DATA_BLOCK "Blok_Bledow"	// DB 119
VERSION : 0.1
  STRUCT
   Blad_Silnika_Adr_1 : BOOL ;	//Blad silnika o adresie 1 - rolki obrotnica bindownicy
   Blad_Silnika_Adr_2 : BOOL ;	//Blad silnika o adresie 2 - rolki wylot bindownicy
   Blad_Silnika_Adr_3 : BOOL ;	//Blad silnika o adresie 3 - rolki
   Blad_Silnika_Adr_4 : BOOL ;	//Blad silnika o adresie 4 - rolki
   Blad_Silnika_Adr_5 : BOOL ;	//Blad silnika o adresie 5 - rolki
   Blad_Silnika_Adr_6 : BOOL ;	//Blad silnika o adresie 6 - rolki
   Blad_Silnika_Adr_7 : BOOL ;	//Blad silnika o adresie 7 - rolki
   Blad_Silnika_Adr_8 : BOOL ;	//Blad silnika o adresie 8 - rolki
   Blad_Silnika_Adr_9 : BOOL ;	//Blad silnika o adresie 9 - rolki
   Blad_Silnika_Adr_10 : BOOL ;	//Blad silnika o adresie 10 - rolki
   Blad_Silnika_Adr_11 : BOOL ;	//Blad silnika o adresie 11 - rolki
   Blad_Silnika_Adr_12 : BOOL ;	//Blad silnika o adresie 12 - rolki
   Blad_Silnika_Adr_13 : BOOL ;	//Blad silnika o adresie 13 - rolki
   Blad_Silnika_Adr_14 : BOOL ;	//Blad silnika o adresie 14 - rolki
   Blad_Silnika_Adr_15 : BOOL ;	//Blad silnika o adresie 15 - silnik obrotnicy bindownicy
   Blad_Rygla_Adr_16 : BOOL ;	//Blad rygla drzwi o adresie 16
   Blad_Silnika_Adr_18 : BOOL ;	//Blad silnika o adresie 18 - silnik obrotnicy wyboru wlotu
   Blad_Silnika_Adr_20 : BOOL ;	//Blad silnika o adresie 20 - silnik obrotnicy etykietownicy
   Blad_Silnika_Adr_23 : BOOL ;	//Blad silnika o adresie 23 - rolki
   Blad_Silnika_Adr_24 : BOOL ;	//Blad silnika o adresie 24 - rolki
   Blad_Kurtyny_Adr_25 : BOOL ;	//Blad kurtyny wlotowej  adres 25
   Blad_Kurtyny_Adr_26 : BOOL ;	//Blad kurtyny wylotowej aders 26
   Blad_Not_Aus_27 : BOOL ;	//Blad Not Aus adres 27 - Not Aus szafa
   Blad_Not_Aus_28 : BOOL ;	//Blad Not Aus adres 28 - Not Aus poczatek lini
   Blad_Not_Aus_29 : BOOL ;	//Blad Not Aus adres 29 - Not Aus srodek lini
   Blad_Not_Aus_30 : BOOL ;	//Blad Not Aus adres 30 - Not Aus koniec lini
   Blad_Not_Aus_31 : BOOL ;	//Blad Not Aus adres 31 - Not Aus panel bindownicy
   Blad_Przek_Bezp_Bind : BOOL ;	//Strefa bezpieczenstwa rejonu bindownicy  niepotwierdzona(wejscie -I4.4)
   Ostrz_Bind_Blad : BOOL ;	//Blad ogolny bindownicy
   Ostrz_Bind_Nie_Cofnieta : BOOL ;	//Bindownica nie jest cofnieta
   Ostrz_Bind_Sygn_Bezp : BOOL ;	//Bindownica brak sygnalu bezpieczenstwa
   Ostrz_Bind_Nie_Jest_Auto : BOOL ;	//Bindownica nie jest w trybie automatycznym (wejscie -I2.4)
   Ostrz_Stol_Obr_Foto : BOOL ;	//Blad fotokomorek stolu obrotowego
   Ostrz_Obr_Stol_Obr_Pozyc : BOOL ;	//Stol obrotowy nie jest w pozycji 0
   Ostrz_Pokr_Foto_Tas_1 : BOOL ;	//Niewlasciwe Pokrycie fotkomorek na tasmie 1 (Przejedz do przodu w recznym )
   Ostrz_Pokr_Foto_Tas_2 : BOOL ;	//Niewlasciwe Pokrycie fotkomorek na tasmie 2 (Przejedz do przodu w recznym )
   Ostrz_Pokr_Foto_Obr : BOOL ;	//Niewlasciwe Pokrycie fotkomorek na obrotnicy (Przejedz do przodu w recznym )
   Ostrz_Pokr_Foto_Tas_4 : BOOL ;	//Niewlasciwe Pokrycie fotkomorek na tasmie 4 (Przejedz do przodu w recznym )
   Blad_Krok_1 : BOOL ;	//Blad kroku nr 1 (Przekrokczony czas jazdy  na zadana pozycje)
   Blad_Krok_2 : BOOL ;	//Blad kroku nr 2 (Przekrokczony czas szukania srodka palety)
   Blad_Krok_3 : BOOL ;	//Blad kroku nr 3 (Przekrokczony czas pozycjonowania palety lewo/prawo)
   Blad_Krok_4 : BOOL ;	//Blad kroku nr 4 (Przekrokczony czas strzalu bindownicy)
   Blad_Krok_5 : BOOL ;	//Blad kroku nr 5 (Przekrokczony czas czasu postoju)
   Blad_Krok_6 : BOOL ;	//Blad kroku nr 6 (Przekrokczony czas powrotu lewo/prawo)
   Alarm_Obr_Stol_Obr_Pozyc : BOOL ;	//Stol obrotowy nie jest w pozycji 0
   Alarm_Bind_Nie_Cofinieta : BOOL ;	//Bindownica nie cofnieta lub brak zezwolenia  (cofnij ramie do tylu)
   Alarm_Bind_Sygn_Bezp : BOOL ;	//Bindownica brak sygnalu bezpieczenstwa
   rez3 : BOOL ;	//rez 3
   rez_6_0 : BOOL ;	//rez_6_0
   Alarm_Pokr_Foto_Tas_1 : BOOL ;	//Niewlasciwe Pokrycie fotkomorek na tasmie 1 (Przejedz do przodu w recznym )
   Alarm_Pokr_Foto_Tas_2 : BOOL ;	//Niewlasciwe Pokrycie fotkomorek na tasmie 2 (Przejedz do przodu w recznym )
   Alarm_Pokr_Foto_Tas_4 : BOOL ;	//Niewlasciwe Pokrycie fotkomorek na tasmie 4 (Przejedz do przodu w recznym )
   Alarm_Pokr_Foto_Obr : BOOL ;	//Niewlasciwe Pokrycie fotkomorek na obrotnicy przy braku cyklu
   Alarm_Bind_Nie_Jest_Auto : BOOL ;	//Bindownica nie jest w trybie automatycznym (wejscie -I2.4)
   Alarm_Bind_Blad : BOOL ;	//Blad ogolny bindownicy
   rez_6_7 : BOOL ;	//rez_6_7
   Ostrz_Prasa_Nie_W_Gorze : BOOL ;	//Zlamywak dekli nie jest u gory I2.6
   rez_7_1 : BOOL ;	//rez_7_1
   rez_7_2 : BOOL ;	//rez_7_2
   rez_7_3 : BOOL ;	//rez_7_3
   rez_7_4 : BOOL ;	//rez_7_4
   rez_7_5 : BOOL ;	//rez_7_5
   Ostrz_Wozek_Przy_Przen : BOOL ;	//Wozek widlowy przy przenosniku (i2.7)
   Ostrz_C_Bind_Foto_Pokr : BOOL ;	//Pokrycie fotokomorek podczas cyklu bindowania
   Ostrz_C_Bind_Poz_Bindow : BOOL ;	//Pozycja bindownicy podczas bindowania
   rez_8_1 : BOOL ;	//rez_8_1
   rez_8_2 : BOOL ;	//rez_8_2
   rez_8_3 : BOOL ;	//rez_8_3
   rez_8_4 : BOOL ;	//rez_8_4
   rez_8_5 : BOOL ;	//rez_8_5
   rez_8_6 : BOOL ;	//rez_8_6
   rez_8_7 : BOOL ;	//rez_8_7
   rez_9_0 : BOOL ;	//rez_9_0
   rez_9_1 : BOOL ;	//rez_9_1
   rez_9_2 : BOOL ;	//rez_9_2
   rez_9_3 : BOOL ;	//rez_9_3
   rez_9_4 : BOOL ;	//rez_9_4
   rez_9_5 : BOOL ;	//rez_9_5
   rez_9_6 : BOOL ;	//rez_9_6
   rez_9_7 : BOOL ;	//rez_9_7
   rez_int_bl : INT ;
   rez_int_bl_2 : INT ;
  END_STRUCT ;	
BEGIN
END_DATA_BLOCK

DATA_BLOCK "DB_HMI"	// DB 120
VERSION : 0.1
  STRUCT
   HMI_IN : STRUCT 	//Zmienne wchodzace do HMI nie nadpisywane W HMI (100 bajtow)
    Tryb_Reczny : BOOL ;	//Tryb Reczny
    Tryb_Auto : BOOL ;	//Tryb Auto
    Pozycja_0_st : BOOL ;	//Obrotnica Pozycja 0 st
    Pozycja_90_st : BOOL ;	//Obrotnica Pozycja 90 st
    Pozycja_180_st : BOOL ;	//Obrotnica Pozycja 180 st
    Pozycja_270_st : BOOL ;	//Obrotnica Pozycja 270 st
    Foto_Tasma_1_Tyl : BOOL ;	//foto tylne na bandzie wlotowej
    Foto_Tasma_1_Przod : BOOL ;	//foto przednie bandzie wlotowej
    Foto_Tasma_2_Tyl : BOOL ;	//foto tylne na bandzie wlotowej 2
    Foto_Tasma_2_Przod : BOOL ;	//foto przednie na bandzie wlotowej 2
    Foto_Obrotnica_3_Tyl : BOOL ;	//foto tylne na obrotnicy 3
    Foto_Obrotnica_3_Przod : BOOL ;	//foto przednie na obrotnicy 3
    Foto_Tasma_4_Tyl : BOOL ;	//foto tylne na bandzie wylotowej 4
    Foto_Tasma_4_Przod : BOOL ;	//foto przednie na bandzie wlotowej 4
    Motor_Tasma_1_Tyl : BOOL ;	//motor tasma 1 tyl
    Motor_Tasma_1_Przod : BOOL ;	//motor tasma 1 przod
    Motor_Tasma_2_Tyl : BOOL ;	//motor tasma 2 tyl
    Motor_Tasma_2_Przod : BOOL ;	//motor tasma 2 przod
    Motor_Tasma_3_Tyl : BOOL ;	//motor tasma obrotnica 3 tyl
    Motor_Tasma_3_Przod : BOOL ;	//motor tasma obrotnica 3 przod
    Motor_Obrotnica_3_CW : BOOL ;	//motor obrotnica 3 clock wise
    Motor_Obrotnica_3_CCW : BOOL ;	//motor obrotnica 3 counter clock wise
    Motor_Tasma_4_Przod : BOOL ;	//motor tasma obrotnica 4 tyl
    Motor_Tasma_4_Tyl : BOOL ;	//motor tasma obrotnica 4 przod
    Kurtyna_Wlot_Ok : BOOL ;	//kurtyna na wlocie ok
    Kurtyna_Wylot_Ok : BOOL ;	//kurtyna na wylocie ok
    Wybrano_TP_Przelot : BOOL ;	//wybrano tryb pracy przelot
    Wybrano_TP_Wiazanie_Wzdl : BOOL ;	//wybrano tryb pracy wiazanie wzdluzne
    Wybrano_TP_Wiazanie_Pop : BOOL ;	//wybrano tryb pracy wiazanie poprzeczne
    Wybrano_TP_Wiazanie_Krzy : BOOL ;	//wybrano tryb pracy wiazanie krzyzowe
    Czujnik_Ham_0_St : BOOL ;	//fotokomorka hamowania obrotnicy do kata 0st
    Czujnik_0_St : BOOL ;	//fotokomorka zatrzymania obrotnicy przy kacie 0st
    Czujnik_Ham_90_St : BOOL ;	//fotokomorka hamowania obrotnicy do kata 90st
    Czujnik_90_St : BOOL ;	//fotokomorka zatrzymania obrotnicy przy kacie 90st
    Czujnik_Ham_180_St : BOOL ;	//fotokomorka hamowania obrotnicy do kata 180st
    Czujnik_180_St : BOOL ;	//fotokomorka zatrzymania obrotnicy przy kacie 180st
    Czujnik_Ham_270_St : BOOL ;	//fotokomorka hamowania obrotnicy do kata 270st
    Czujnik_270_St : BOOL ;	//fotokomorka zatrzymania obrotnicy przy kacie 270st
    Interfefs_B_do_TP_B1 : BOOL ;	//obwod bezpieczenstwa bindownicy
    Interfefs_B_do_TP_B2 : BOOL ;	//polozenie podstawowe bindownicy
    Interfefs_B_do_TP_B3 : BOOL ;	//start/zakonczenie wiazania
    Interfefs_B_do_TP_B5 : BOOL ;	//blad bindownicy
    Interfefs_TP_do_B_TP1 : BOOL ;	//obwod bezpieczenstwa tasmociagow
    Interfefs_TP_do_B_TP2 : BOOL ;	//zezwolenie na prace bindownicy
    Interfefs_TP_do_B_TP3 : BOOL ;	//start wiazania
    PB_Strefa_bezpieczenstwa : BOOL ;	//przycisk zalaczenie Strefy bezpieczenstwa
    PB_Reczny : BOOL ;	//przycisk trybu reczny
    PB_Auto : BOOL ;	//przycisk auto
    PB_Reset : BOOL ;	//przycisk reset
    PB_Stop : BOOL ;	//przycisk stop
    PB_Cykl_Start : BOOL ;	//przycisk start cyklu
    PB_Tasma1_Tyl : BOOL ;	//przycisk tasma 1 do tylu
    PB_Tasma1_Przod : BOOL ;	//przycisk tasma 1 do przodu
    PB_Tasma2_Tyl : BOOL ;	//przycisk tasma 2 do tylu
    PB_Tasma2_Przod : BOOL ;	//przycisk tasma 2 do przodu
    PB_Tasma3_Tyl : BOOL ;	//przycisk tasma 3 do tylu
    PB_Tasma3_Przod : BOOL ;	//przycisk tasma 3 do przodu
    PB_Tasma4_Tyl : BOOL ;	//przycisk tasma 4 do tylu
    PB_Tasma4_Przod : BOOL ;	//przycisk tasma 4 do przodu
    PB_Tasma3_Obr_CW : BOOL ;	//przycisk obrotnica w prawo
    PB_Tasma3_Obr_CCW : BOOL ;	//przycisk obrotnica w lewo
    Lampka_Blad_Bind : BOOL ;	//lamka bledu bindownicy
    Lampka_Strzal_Tasmy : BOOL ;	//lampka wystrzalu tasmy
    Lampka_Strefa_Bezp : BOOL ;	//lampka przycisku strefy bezpieczenstwa
    Lampka_PB_Reczny : BOOL ;	//lampka przycisku trybu recznego
    Lampka_PB_Auto : BOOL ;	//lampka przycisku trybu auto
    Lampka_PB_Reset : BOOL ;	//lampka przycisku reset
    Lampka_PB_Stop : BOOL ;	//lampka przycisku stop
    Lampka_PB_Cykl_Start : BOOL ;	//lampka przycisku start
    Paleta_na_Tasmie_1 : BOOL ;	//znacznik palety na tasmie 1
    Paleta_na_Tasmie_2 : BOOL ;	//znacznik palety na tasmie 2
    Paleta_na_Tasmie_3_0_180 : BOOL ;	//znacznik palety na tasmie 3 przy kacie 0 lub 180st
    Paleta_na_Tasmie_3_90_27 : BOOL ;	//znacznik palety na tasmie 3 przy kacie 90 lub 270st
    Paleta_na_Tasmie_4 : BOOL ;	//znacznik palety na tasmie 4
    Paleta_na_Tasmie_1_T : BOOL ;	//znacznik palety na tasmie 1 wjazd
    Paleta_na_Tasmie_1_P : BOOL ;	//znacznik palety na tasmie 1 wyjazd
    Paleta_na_Tasmie_2_T : BOOL ;	//znacznik palety na tasmie 2 wjazd
    Paleta_na_Tasmie_2_P : BOOL ;	//znacznik palety na tasmie 2 wyjazd
    Paleta_na_Tasmie_3_T : BOOL ;	//znacznik palety na tasmie 3 wjazd
    Paleta_na_Tasmie_3_P : BOOL ;	//znacznik palety na tasmie 3 wyjazd
    Paleta_na_Tasmie_4_T : BOOL ;	//znacznik palety na tasmie 4 wjazd
    Paleta_na_Tasmie_4_P : BOOL ;	//znacznik palety na tasmie 4 wyjazd
    Rygiel : BOOL ;	//znacznik rygla drzwi
    Blad : BOOL ;	//Znacznik bledu
    Linia_transportowa_praca : BOOL ;	//Znacznik pracy calej linii transportowej
    Interfefs_B_do_TP_B4 : BOOL ;	//tryb pracy bindownicy: Auto(1) Reczny(0)
    Krok_1 : BOOL ;	//krok 1 trybu pracy
    Krok_2 : BOOL ;	//krok 2 trybu pracy
    Krok_3 : BOOL ;	//krok 3 trybu pracy
    Krok_4 : BOOL ;	//krok 4 trybu pracy
    Krok_5 : BOOL ;	//krok 5 trybu pracy
    Krok_6 : BOOL ;	//krok 6 trybu pracy
    Znacznik_Migania_Bledu : BOOL ;	//znacznik migania bledu
    Czujnik_Prasa : BOOL ;	//czujnik prasy s 22
    Stan_Zaworu : BOOL ;
    Gender_Jest_Online : BOOL ;	//Zalacz Gender do lini Gender Feeder
    Gender_Jest_OFFline : BOOL ;	//Odlacz Gender do lini Gender Feeder
    Obr_Gender_Wzdluz : BOOL ;
    Obr_za_Genderem_wzdluz : BOOL ;
    Obr_za_Foliarka_wzdluz : BOOL ;
    Obr_Gender_ukryj : BYTE ;
    Obr_za_Genderem_ukryj : BYTE ;
    Obr_za_Foliarka_ukryj : BYTE ;
    Tablica_IN_bool : ARRAY  [1 .. 10 ] OF BOOL  := FALSE;
    Tablica_IN_Byte : ARRAY  [1 .. 2 ] OF BYTE  := B#16#0;
    input_0 : BYTE ;
    input_1 : BYTE ;
    input_2 : BYTE ;
    input_3 : BYTE ;
    output_0 : BYTE ;
    output_1 : BYTE ;
    output_2 : BYTE ;
    output_3 : BYTE ;
    input_8 : BYTE ;
    input_9 : BYTE ;
    input_10 : BYTE ;
    input_11 : BYTE ;
    Tablica_IN_DWORD : ARRAY  [1 .. 4 ] OF DWORD ;
    NR_Kroku : DINT ;	//Numer kroku
    Aktualna_Data : DATE_AND_TIME ;
    Tablica_IN_INT : ARRAY  [1 .. 18 ] OF INT ;
    tryb_wiaz : INT ;	//znacznik wyboru trybu wiazania
    INT_Liczba_Akt_Kroku : INT ;	//znacznik wyboru aktualnie wykonywanego kroku
   END_STRUCT ;
   HMI_OUT : STRUCT 	//Zmienne wychodzace z HMI Nie nadpisywane w sterowniku od 100 bajta
    Wybor_2_Lap : BOOL ;	//Wybranie 2 lap
    Wybor_4_Lap : BOOL ;	//Wybranie 4 lap
    Start_Lini_z_OP : BOOL ;	//start calej lini z HMI
    Stop_Lini_z_OP : BOOL ;	//stop calej lini z HMI
    Wyzwolenie_Wyjazdu : BOOL ;	//wyzwolenie wyjazdu palety na stanowisku bindujacym (tylko w auto)
    Przycisk_Test_Lampek : BOOL ;	//przycisk test lampek
    Przycisk_Reset_Bledow : BOOL ;	//Przycisk resetowania bledow na panelu HMI
    Przycisk_Pozycjonowanie : BOOL ;	//Przycisk HMI do pozycjonowania palety
    H_Zalacz_Zawor_Prasa : BOOL ;	//Zalacz zawor prasa
    H_Zezwl_Ekran_Prasa : BOOL ;	//Zezwolenie na prase reczny
    PB_Gender_ONline : BOOL ;	//Przycisk Gender jest online z linia transportowa
    PB_Gender_OFFline : BOOL ;	//Przycisk Gender jest offline z linia transportowa
    Tablica_OUT_Bool : ARRAY  [1 .. 144 ] OF BOOL ;
    Tablina_OUT_INT : ARRAY  [1 .. 40 ] OF INT ;
   END_STRUCT ;
   HMI_IN_OUT : STRUCT 	//Zmienne nadpisywane w sterowniku i w HMI od 200 bajta
    Rezerwa_IN_Out_1 : BOOL ;
    Tp_Przelot : BOOL ;	//Tryb Pracy Przelot
    Tp_Wiazanie_Poprzeczne : BOOL ;	//Tryb Pracy Wiazanie poprzeczne
    Tp_Wiazanie_Wzdluzne : BOOL ;	//Tryb Pracy Wiazanie wzduzne
    Tp_Wiazanie_Pop_Wzdl : BOOL ;	//Tryb Pracy Wiaznie Poprzeczne i wzdluzne
    Tp_Pozycjonowanie : BOOL ;	//Tryb Pracy Pozycjonowanie Palety zalaczone
    Test_Lampek : BOOL ;	//Test Lampek
    Reset_bledow : BOOL ;	//Reset Bledow
    Zlamywak_Dekl : BOOL ;	//lamanie dekli
    Tablica_IN_OUT_Bool : ARRAY  [1 .. 144 ] OF BOOL ;
    Tablica_IN_OUT_INT : ARRAY  [1 .. 40 ] OF INT ;
    Wybor_trybu_pracy : BYTE ;
   END_STRUCT ;
  END_STRUCT ;	
BEGIN
   HMI_IN.Foto_Obrotnica_3_Przod := TRUE;
   HMI_IN.Czujnik_0_St := TRUE;
END_DATA_BLOCK

DATA_BLOCK "Kom_Shuttle"	// DB 205
VERSION : 0.1
  STRUCT
   OUT : STRUCT 	//Temporary placeholder variable
    Bit_Com_Odbieranie : BOOL ;
    Auto_Reczny_Gender : BOOL ;	//1-auto , 0- reczny
    Marka_Bezp_Gender : BOOL ;
    Linia_Gender_Online : BOOL ;	//Linia Gender odbiera palety z shuttle
    Blad_Lini_Gender : BOOL ;	//Linia Gender jest w bledzie
    Res_0_5 : BOOL ;
    PB_Auto : BOOL ;
    PB_Reczny : BOOL ;
    PB_Banda_Wozek_Przod : BOOL ;
    PB_Banda_Wozek_Tyl : BOOL ;
    Banda_1_Gen_Zez_Do_Pop : BOOL ;	//banda gender zezwolenie do porzedniej
    Banda_1_Gen_Pal_Dost : BOOL ;	//Paleta dostarczona
    Banda_1_Gen_Zez_R_Do_Pop : BOOL ;	//zezwolenie reczny do poprzedniej
    Res_1_5 : BOOL ;
    Res_1_6 : BOOL ;
    Res_1_7 : BOOL ;
    Bindownica_Agregat_Auto : BOOL ;	//Agregat bindownicy jest w auto
    Res_2_1 : BOOL ;
    Res_2_2 : BOOL ;
    Res_2_3 : BOOL ;
    Res_2_4 : BOOL ;
    Res_2_5 : BOOL ;
    Res_2_6 : BOOL ;
    Res_2_7 : BOOL ;
    Res_3_0 : BOOL ;
    Res_3_1 : BOOL ;
    Res_3_2 : BOOL ;
    Res_3_3 : BOOL ;
    Res_3_4 : BOOL ;
    Res_3_5 : BOOL ;
    Res_3_6 : BOOL ;
    Res_3_7 : BOOL ;
    Zmienna_DINT : DINT ;
   END_STRUCT ;
   IN : STRUCT 	//Temporary placeholder variable
    Bit_Com_Odbieranie : BOOL ;
    Auto_Reczny_Shuttle : BOOL ;	//1-auto , 0- reczny
    Marka_Bezp_Shuttle : BOOL ;
    Wymuszenie_Online : BOOL ;	//Wymuszenie Lini gender online
    Wymuszenie_Offline : BOOL ;	//Wymuszenie Lini gender offline (wykorzystanie wozka widlowego)
    Wozek_Na_Pozycji_Gender : BOOL ;	//Wozek znajduje sie na pozycji
    Wozek_Zasprzeglony : BOOL ;
    Res_0_7 : BOOL ;	//Przycisk reczny
    Wozek_Zab_do_Nast : BOOL ;	//Wozek zabierz do nastepnej
    Wozek_Zez_R_do_Nast : BOOL ;	//Wozek zezwolenie reczny do nastepnej
    Foto_Wozek_Przod : BOOL ;	//Foto Wozek Przod
    Foto_Wozek_Tyl : BOOL ;	//Foto Wozek Tyl
    Motor_Wozek_Tyl : BOOL ;	//Motor wozek tyl
    Motor_Wozek_Przod : BOOL ;	//Motor wozek przod
    Res_1_6 : BOOL ;
    Res_1_7 : BOOL ;
    Res_2_0 : BOOL ;
    Res_2_1 : BOOL ;
    Res_2_2 : BOOL ;
    Res_2_3 : BOOL ;
    Res_2_4 : BOOL ;
    Res_2_5 : BOOL ;
    Res_2_6 : BOOL ;
    Res_2_7 : BOOL ;
    Res_3_0 : BOOL ;
    Res_3_1 : BOOL ;
    Res_3_2 : BOOL ;
    Res_3_3 : BOOL ;
    Res_3_4 : BOOL ;
    Res_3_5 : BOOL ;
    Res_3_6 : BOOL ;
    Res_3_7 : BOOL ;
    Zmienna_DINT : DINT ;
   END_STRUCT ;
  END_STRUCT ;	
BEGIN
END_DATA_BLOCK

DATA_BLOCK "Rejestr Band"	// DB 310
VERSION : 0.1
  STRUCT
   Tasma_Wozek_0 : DINT ;	//Wartosc tasmy wozek
   Tasma_Gender_1 : DINT ;	//Wartosc tasmy gender
   Tasma_Gender_2 : DINT ;	//Wartosc tasmy gender
   Tasma_Gender_Obr_3 : DINT ;	//Wartosc tasmy gender obrot
   Tasma_Gender_4 : DINT ;	//Wartosc tasmy gender wylot
   Tasma_Transp_Obr_4 : DINT ;	//Wartosc tasmy obrotnicy 1 transportera
   Tasma_Transp_3 : DINT ;	//Tasma transportowa wlot 2
   Tasma_Transp_5 : DINT ;	//Tasma transportowa 5
   Tasma_Transp_6 : DINT ;	//Tasma transportowa 6
   Tasma_Transp_7 : DINT ;	//Tasma transportowa 7
   Tasma_Transp_8 : DINT ;	//Tasma transportowa 8
   Tasma_Transp_9 : DINT ;	//Tasma transportowa 9
   Tasma_Transp_10_Fol : DINT ;	//Tasma transportowa 10 wspolnsna z foliarka
   Tasma_Transp_4_Fol : DINT ;	//Tasma transportowa virtual 4
   Tasma_Transp_Obr_Fol : DINT ;	//Tasma transportowa obrotnica virtual 5
   Tasma_Transp_6_Fol : DINT ;	//Tasma za obrotnica virtulal 6
   Tasma_Transp_11_Fol : DINT ;	//Tasma transportowa 11 wspolna z foliarka
   Tasma_Transp_12 : DINT ;	//Tasma transportowa wlot 12
   Tasma_Transp_Obr_13 : DINT ;	//Tasma transportowa 13 obrotnica
   Tasma_Wysjsciowa_14 : DINT ;	//Tasma transportowa 14 wylot
  END_STRUCT ;	
BEGIN
END_DATA_BLOCK

DATA_BLOCK "Rejestr_Band_HMI"	// DB 311
VERSION : 0.1
  STRUCT
   Tasma_Wozek_0_HMI : DINT ;	//Wartosc tasmy wozek
   Tasma_Gender_1_HMI : DINT ;	//Wartosc tasmy gender
   Tasma_Gender_2_HMI : DINT ;	//Wartosc tasmy gender
   Tasma_Gender_Obr_3_HMI : DINT ;	//Wartosc tasmy gender obrot
   Tasma_Gender_4_HMI : DINT ;	//Wartosc tasmy gender wylot
   Tasma_Transp_Obr_4_HMI : DINT ;	//Wartosc tasmy obrotnicy 1 transportera
   Tasma_Transp_3_HMI : DINT ;	//Tasma transportowa wlot 2
   Tasma_Transp_5_HMI : DINT ;	//Tasma transportowa 5
   Tasma_Transp_6_HMI : DINT ;	//Tasma transportowa 6
   Tasma_Transp_7_HMI : DINT ;	//Tasma transportowa 7
   Tasma_Transp_8_HMI : DINT ;	//Tasma transportowa 8
   Tasma_Transp_9_HMI : DINT ;	//Tasma transportowa 9
   Tasma_Transp_10_Fol_HMI : DINT ;	//Tasma transportowa 10 wspolnsna z foliarka
   Tasma_Transp_4_Fol_HMI : DINT ;	//Tasma transportowa virtual 4
   Tasma_Transp_Obr_Fol_HMI : DINT ;	//Tasma transportowa obrotnica virtual 5
   Tasma_Transp_6_Fol_HMI : DINT ;	//Tasma za obrotnica virtulal 6
   Tasma_Transp_11_Fol_HMI : DINT ;	//Tasma transportowa 11 wspolna z foliarka
   Tasma_Transp_12_HMI : DINT ;	//Tasma transportowa wlot 12
   Tasma_Transp_Obr_13_HMI : DINT ;	//Tasma transportowa 13 obrotnica
   Tasma_Wysjsciowa_14_HMI : DINT ;	//Tasma transportowa 14 wylot
  END_STRUCT ;	
BEGIN
END_DATA_BLOCK

ORGANIZATION_BLOCK OB 1
TITLE = "Main Program Sweep (Cycle)"
VERSION : 0.1
VAR_TEMP
  OB1_EV_CLASS : BYTE ;	//Bits 0-3 = 1 (Coming event), Bits 4-7 = 1 (Event class 1)
  OB1_SCAN_1 : BYTE ;	//1 (Cold restart scan 1 of OB 1), 3 (Scan 2-n of OB 1)
  OB1_PRIORITY : BYTE ;	//Priority of OB Execution
  OB1_OB_NUMBR : BYTE ;	//1 (Organization block 1, OB1)
  OB1_RESERVED_1 : BYTE ;	//Reserved for system
  OB1_RESERVED_2 : BYTE ;	//Reserved for system
  OB1_PREV_CYCLE : INT ;	//Cycle time of previous OB1 scan (milliseconds)
  OB1_MIN_CYCLE : INT ;	//Minimum cycle time of OB1 (milliseconds)
  OB1_MAX_CYCLE : INT ;	//Maximum cycle time of OB1 (milliseconds)
  OB1_DATE_TIME : DATE_AND_TIME ;	//Date and time OB1 started
END_VAR
BEGIN
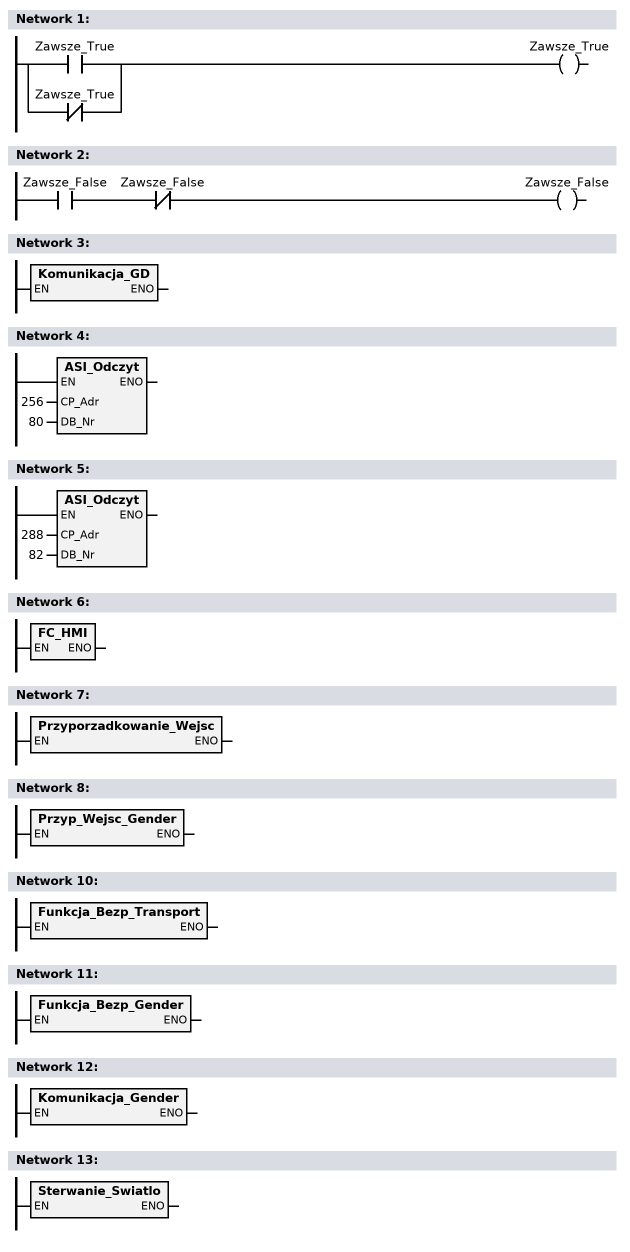
NETWORK
TITLE =
//Zawsze true
      O     "Zawsze_True";
      ON    "Zawsze_True";
      =     "Zawsze_True";
NETWORK
TITLE =
//Zawsze False
      A     "Zawsze_False";
      AN    "Zawsze_False";
      =     "Zawsze_False";
NETWORK
TITLE =
//   BEU   
      CALL  "Komunikacja_GD";
      NOP   0;
NETWORK
TITLE =
//Odczyt wejsc ASI Transporter
//
      CALL  "ASI_Odczyt" (
           CP_Adr                   := 256,
           DB_Nr                    := 80);
      NOP   0;
NETWORK
TITLE =
//Odczyt Wejsc Asi Gender
      CALL  "ASI_Odczyt" (
           CP_Adr                   := 288,
           DB_Nr                    := 82);
      NOP   0;
NETWORK
TITLE =
//komunikacja z hmi
      CALL  "FC_HMI";
      NOP   0;
NETWORK
TITLE =
      CALL  "Przyporzadkowanie_Wejsc";
      NOP   0;
NETWORK
TITLE =
      CALL  "Przyp_Wejsc_Gender";
      NOP   0;
NETWORK
TITLE =
NETWORK
TITLE =
      CALL  "Funkcja_Bezp_Transport";
      NOP   0;
NETWORK
TITLE =
      CALL  "Funkcja_Bezp_Gender";
      NOP   0;
NETWORK
TITLE =
      CALL  "Komunikacja_Gender";
      NOP   0;
NETWORK
TITLE =
      CALL  "Sterwanie_Swiatlo";
      NOP   0;
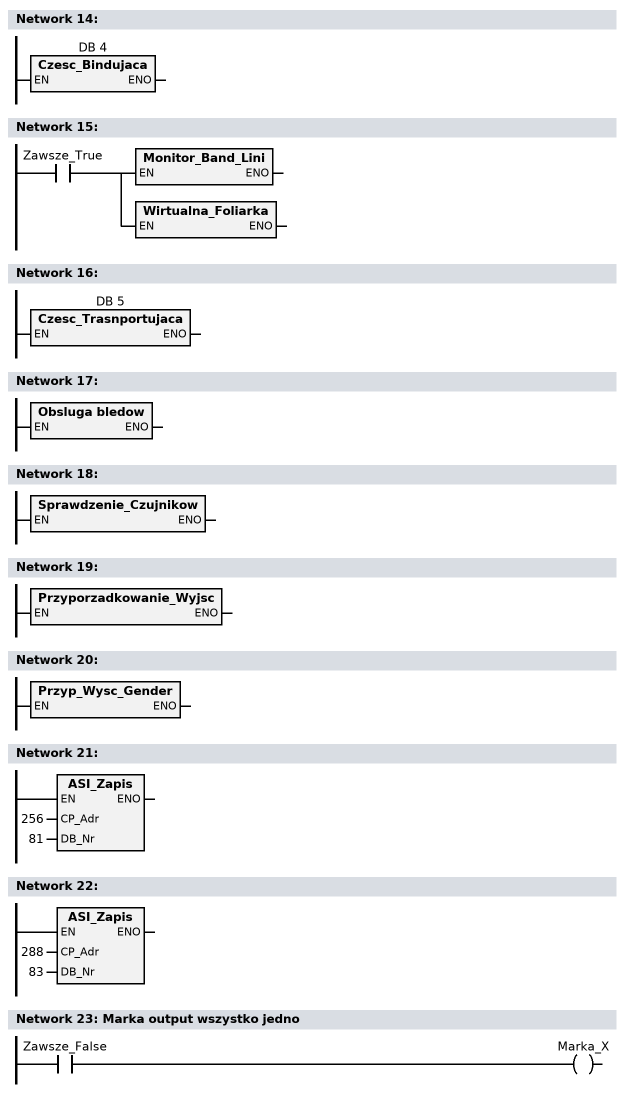
NETWORK
TITLE =
      CALL  "Czesc_Bindujaca" , DB 4;
      NOP   0;
NETWORK
TITLE =
      A     "Zawsze_True";
      =     L 20.0;
      A     L 20.0;
      JNB   _001;
      CALL  "Monitor_Band_Lini";
_001: NOP   0;
      A     L 20.0;
      JNB   _002;
      CALL  "Wirtualna_Foliarka";
_002: NOP   0;
NETWORK
TITLE =
      CALL  "Czesc_Trasnportujaca" , DB 5;
      NOP   0;
NETWORK
TITLE =
      CALL  "Obsluga bledow";
      NOP   0;
NETWORK
TITLE =
      CALL  "Sprawdzenie_Czujnikow";
      NOP   0;
NETWORK
TITLE =
      CALL  "Przyporzadkowanie_Wyjsc";
      NOP   0;
NETWORK
TITLE =
      CALL  "Przyp_Wysc_Gender";
      NOP   0;
NETWORK
TITLE =
//Zapis wyjs Asi Transporter
      CALL  "ASI_Zapis" (
           CP_Adr                   := 256,
           DB_Nr                    := 81);
      NOP   0;
NETWORK
TITLE =
//Zapis wyjsc gender 
      CALL  "ASI_Zapis" (
           CP_Adr                   := 288,
           DB_Nr                    := 83);
      NOP   0;
NETWORK
TITLE = Marka output wszystko jedno
      A     "Zawsze_False";
      =     "Marka_X";
NETWORK
TITLE =
END_ORGANIZATION_BLOCK

ORGANIZATION_BLOCK "I/O_FLT1"	// OB 82
TITLE = "I/O Point Fault"
VERSION : 0.1
VAR_TEMP
  OB82_EV_CLASS : BYTE ;	//16#39, Event class 3, Entering event state, Internal fault event
  OB82_FLT_ID : BYTE ;	//16#XX, Fault identifcation code
  OB82_PRIORITY : BYTE ;	//Priority of OB Execution
  OB82_OB_NUMBR : BYTE ;	//82 (Organization block 82, OB82)
  OB82_RESERVED_1 : BYTE ;	//Reserved for system
  OB82_IO_FLAG : BYTE ;	//Input (01010100), Output (01010101)
  OB82_MDL_ADDR : WORD ;	//Base address of module with fault
  OB82_MDL_DEFECT : BOOL ;	//Module defective
  OB82_INT_FAULT : BOOL ;	//Internal fault
  OB82_EXT_FAULT : BOOL ;	//External fault
  OB82_PNT_INFO : BOOL ;	//Point information
  OB82_EXT_VOLTAGE : BOOL ;	//External voltage low
  OB82_FLD_CONNCTR : BOOL ;	//Field wiring connector missing
  OB82_NO_CONFIG : BOOL ;	//Module has no configuration data
  OB82_CONFIG_ERR : BOOL ;	//Module has configuration error
  OB82_MDL_TYPE : BYTE ;	//Type of module
  OB82_SUB_MDL_ERR : BOOL ;	//Sub-Module is missing or has error
  OB82_COMM_FAULT : BOOL ;	//Communication fault
  OB82_MDL_STOP : BOOL ;	//Module is stopped
  OB82_WTCH_DOG_FLT : BOOL ;	//Watch dog timer stopped module
  OB82_INT_PS_FLT : BOOL ;	//Internal power supply fault
  OB82_PRIM_BATT_FLT : BOOL ;	//Primary battery is in fault
  OB82_BCKUP_BATT_FLT : BOOL ;	//Backup battery is in fault
  OB82_RESERVED_2 : BOOL ;	//Reserved for system
  OB82_RACK_FLT : BOOL ;	//Rack fault, only for bus interface module
  OB82_PROC_FLT : BOOL ;	//Processor fault
  OB82_EPROM_FLT : BOOL ;	//EPROM fault
  OB82_RAM_FLT : BOOL ;	//RAM fault
  OB82_ADU_FLT : BOOL ;	//ADU fault
  OB82_FUSE_FLT : BOOL ;	//Fuse fault
  OB82_HW_INTR_FLT : BOOL ;	//Hardware interupt input in fault
  OB82_RESERVED_3 : BOOL ;	//Reserved for system
  OB82_DATE_TIME : DATE_AND_TIME ;	//Date and time OB82 started
END_VAR
BEGIN
// (block stored without names or comments; labels and parameter names are numbered)
END_ORGANIZATION_BLOCK

ORGANIZATION_BLOCK "RACK_FLT"	// OB 86
TITLE = "Loss Of Rack Fault"
VERSION : 0.1
VAR_TEMP
  OB86_EV_CLASS : BYTE ;	//16#38/39 Event class 3
  OB86_FLT_ID : BYTE ;	//16#C1/C4/C5, Fault identifcation code
  OB86_PRIORITY : BYTE ;	//Priority of OB Execution
  OB86_OB_NUMBR : BYTE ;	//86 (Organization block 86, OB86)
  OB86_RESERVED_1 : BYTE ;	//Reserved for system
  OB86_RESERVED_2 : BYTE ;	//Reserved for system
  OB86_MDL_ADDR : WORD ;	//Base address of IM module in rack with fault
  OB86_RACKS_FLTD : ARRAY  [0 .. 31 ] OF BOOL ;	//Racks in fault
  OB86_DATE_TIME : DATE_AND_TIME ;	//Date and time OB86 started
END_VAR
BEGIN
// (block stored without names or comments; labels and parameter names are numbered)
END_ORGANIZATION_BLOCK

ORGANIZATION_BLOCK "COMPLETE RESTART"	// OB 100
TITLE = "Complete Restart"
VERSION : 0.1
VAR_TEMP
  OB100_EV_CLASS : BYTE ;	//16#13, Event class 1, Entering event state, Event logged in diagnostic buffer
  OB100_STRTUP : BYTE ;	//16#81/82/83/84 Method of startup
  OB100_PRIORITY : BYTE ;	//Priority of OB Execution
  OB100_OB_NUMBR : BYTE ;	//100 (Organization block 100, OB100)
  OB100_RESERVED_1 : BYTE ;	//Reserved for system
  OB100_RESERVED_2 : BYTE ;	//Reserved for system
  OB100_STOP : WORD ;	//Event that caused CPU to stop (16#4xxx)
  OB100_STRT_INFO : DWORD ;	//Information on how system started
  OB100_DATE_TIME : DATE_AND_TIME ;	//Date and time OB100 started
END_VAR
BEGIN
NETWORK
TITLE =
END_ORGANIZATION_BLOCK

ORGANIZATION_BLOCK "PROG_ERR"	// OB 121
TITLE = "Programming Error"
VERSION : 0.1
VAR_TEMP
  OB121_EV_CLASS : BYTE ;	//16#25, Event class 2, Entering event state, Internal fault event
  OB121_SW_FLT : BYTE ;	//16#XX Software programming fault
  OB121_PRIORITY : BYTE ;	//Priority of OB Execution
  OB121_OB_NUMBR : BYTE ;	//121 (Organization block 121, OB121)
  OB121_BLK_TYPE : BYTE ;	//16#88/8A/8B/8C/8E Type of block fault occured in
  OB121_RESERVED_1 : BYTE ;	//Reserved for system
  OB121_FLT_REG : WORD ;	//16#XX Specific register that caused fault
  OB121_BLK_NUM : WORD ;	//Number of block that programming fault occured in
  OB121_PRG_ADDR : WORD ;	//Address in block where programming fault occured
  OB121_DATE_TIME : DATE_AND_TIME ;	//Date and time OB121 started
END_VAR
BEGIN
// (block stored without names or comments; labels and parameter names are numbered)
END_ORGANIZATION_BLOCK

ORGANIZATION_BLOCK "MOD_ERR"	// OB 122
TITLE = "Module Access Error"
VERSION : 0.1
VAR_TEMP
  OB122_EV_CLASS : BYTE ;	//16#29, Event class 2, Entering event state, Internal fault event
  OB122_SW_FLT : BYTE ;	//16#XX Software error code
  OB122_PRIORITY : BYTE ;	//Priority of OB Execution
  OB122_OB_NUMBR : BYTE ;	//122 (Organization block 122, OB122)
  OB122_BLK_TYPE : BYTE ;	//16#88/8C/8E Type of block fault occured in
  OB122_MEM_AREA : BYTE ;	//Memory area where access error occured
  OB122_MEM_ADDR : WORD ;	//Memory address where access error occured
  OB122_BLK_NUM : WORD ;	//Block number in which error occured
  OB122_PRG_ADDR : WORD ;	//Program address where error occured
  OB122_DATE_TIME : DATE_AND_TIME ;	//Date and time OB1 started
END_VAR
BEGIN
// (block stored without names or comments; labels and parameter names are numbered)
END_ORGANIZATION_BLOCK

SYMBOL_TABLE
"Instancja_FB1"	DB 1	FB 1
"Instancja_FB3"	DB 3	FB 3
"Instancja_FB4"	DB 4	FB 4
"DB_CONECTOR"	DB 10	DB 10	// Blok porzadkujacy czujniki lini
"DB_CONECTOR_KB1"	DB 11	DB 11
"DB_CONECTOR_KB2"	DB 12	DB 12
"DB_CONNECTOR_BUFF"	DB 13	DB 13
"DB_CONNECTOR_GEN"	DB 14	DB 14
"Asi_input"	DB 80	DB 80
"Asi_output"	DB 81	DB 81
"DB_ASI_Prosty_Odczyt_KB1"	DB 82	DB 82	// KB1
"DB_ASI_Prosty_Zapis_KB1"	DB 83	DB 83
"DB_ASI_Prosty_Odczyt_KB2"	DB 84	DB 84
"DB_ASi_Prosty_Zapis_KB2"	DB 85	DB 85
"DB_ASi_Prosty_Odczyt_Buf"	DB 86	DB 86	// Odczyt buffory
"DB_ASi_Prosty_Zapis_Buf"	DB 87	DB 87	// Asi db buffory
"Bledy_Shuttle"	DB 116	DB 116
"Bledy_KB1"	DB 117	DB 117
"Bledy_KB2"	DB 118	DB 118
"Bledy_Buffor"	DB 119	DB 119
"DB_HMI_KB1"	DB 121	DB 121
"DB_HMI_KB2"	DB 122	DB 122
"DB_HMI_BUF"	DB 123	DB 123
"DB_HMI_Wozek"	DB 128	DB 128
"COM_SHUTTLE"	DB 200	DB 200	// Blok komunikacji odbieranie shuttle
"LLOUT"	DB 201	DB 201
"LLIN"	DB 202	DB 202	// Blok wymiany danych dlugi
"COM_GENDER"	DB 205	DB 205
"Stale_Maszynowe"	DB 300	DB 300
"DB_Trace"	DB 402	DB 402
"Key_DB"	DB 409	DB 409
"Blok_Default"	DB 800	DB 800
"Blok_Write"	DB 801	DB 801
"Blok_Read"	DB 802	DB 802
"Def_Blok_Para_Wozek"	DB 811	DB 811
"Def_Blok_Kier_KB1"	DB 820	DB 820	// Blok stref kierunek KB1
"Def_Blok_Kier_Rot"	DB 821	DB 821
"Buffor_Rejestr"	DB 823	DB 823
"Buffor_Rejestr_HMI"	DB 824	DB 824
"Def_Stale_Maszynowe"	DB 830	DB 830
"Buffor_Kolejka"	DB 1123	DB 1123
"Blok_Def_Parametry"	DB 1701	DB 1701	// Blok Defaultowy parametrow
"Blok_Parametrow"	DB 1702	DB 1702
"Blok_Def_Kier_KB1"	DB 1720	DB 1720
"Blok_Def_Kier_Rot"	DB 1721	DB 1721
"Stan_Shuttle"	FB 1	FB 1
"Stanowisko_KB1"	FB 3	FB 3	// Stanowisko Kolbus 1
"Stanowisko_KB2"	FB 4	FB 4	// Stanowisko Kolbus 2
"Blok_Jazdy_Band"	FB 5	FB 5
"Stan_Intro_Odbieranie"	FB 6	FB 6
"Stan_Intro_Pob_I1"	FB 7	FB 7
"Stan_Intro_Pob_I2"	FB 8	FB 8	// Stanowisko wozek jezdny
"Stan_Intro_Pob_I3"	FB 9	FB 9
"FB_Uzbrajanie"	FB 10	FB 10	// Funkcja uzbrajanie\
"Filtr_zbocza_2"	FB 14	FB 14
"T_ON"	FB 20	FB 20	// Timer on delay with memory
"T_ON_+_RESET"	FB 21	FB 21	// Czasowka on delay z zapamietanym czasem  + reset
"Banda_Pojedyncza"	FB 30	FB 30
"Banda_Obr_1"	FB 31	FB 31	// Banda obrotowa o dwoch wlotach i jednej fotokomorce
"Band_Wozka"	FB 32	FB 32	// Banda wozka z trybem recznym
"Banda_Poj_+_Tryb_Reczny"	FB 33	FB 33
"B_Obr_+_Reczny"	FB 35	FB 35
"Banda_Obr_+_Reczny"	FB 36	FB 36	// Banda obrotwa + reczny
"Banda_Poj_+_Winda"	FB 37	FB 37	// Banda pojedyncza + winda + tryb reczny
"Wybranie_Wjazdu"	FB 50	FB 50
"Obr_Na_Poz_1"	FB 51	FB 51
"Pozycjonowanie_Bandy"	FB 55	FB 55
"Obr_Na_Poz_1_Pelny"	FB 61	FB 61
"KB2_Reczny"	FC 1	FC 1
"Funkcja_Bezpieczenstwa"	FC 3	FC 3
"Oryginalna_FC3"	FC 4	FC 4
"Wozek_Jezdny_Jazda"	FC 5	FC 5
"Wozek_Jezdny_Jazda_2"	FC 6	FC 6	// Funkcja sterujaca lampkami
"Sprawdzenie_Okna"	FC 7	FC 7	// Sprawdzenie czy wartosc miesci sie w oknie
"Lenze_Sew_Shell_KB1"	FC 8	FC 8
"Lenze_Sew_Shell_KB2"	FC 9	FC 9	// Nakladka na falownik Lenze by czytac jak Sewa
"Fal_Lenze_V_3"	FC 10	FC 10
"Przyciski_Dwufunkcyjne"	FC 11	FC 11
"Sterowanie_Ramp"	FC 12	FC 12
"Auto_Reczny_KB1"	FC 13	FC 13
"Auto_Reczny_KB2"	FC 14	FC 14
"Auto_Reczny_Buff"	FC 15	FC 15
"Przyporzadkowanie_Wejsc"	FC 20	FC 20
"Przyporzadkowanie_Wyjsc"	FC 21	FC 21
"Przypis_Wejsc_KB1"	FC 22	FC 22
"Przypis_Wyjsc_KB1"	FC 23	FC 23
"Przypis_Wejsc_KB2"	FC 24	FC 24
"Przypis_Wyjsc_KB2"	FC 25	FC 25
"Przypis_Wejsc_Buffory"	FC 26	FC 26
"Przypis_Wyjsc_Buffory"	FC 27	FC 27
"Rejestr_Tasm"	FC 30	FC 30
"qqq"	FC 31	FC 31
"Ruch_Palety"	FC 40	FC 40
"Ruch_Palety_Winda"	FC 41	FC 41	// Kasowanie_Bledow
"Wybor_Wjazdu"	FC 50	FC 50	// Wybor miejsca pobierania palety
"Obrotnica_Na_Pozycje"	FC 51	FC 51
"LT_BT"	FC 62	FC 62	// Convert local time to base time
"ASI_Odczyt"	FC 80	FC 80
"ASI_Zapis"	FC 81	FC 81
"ASI_Prosty_Odczyt"	FC 82	FC 82	// Prosty odczyt modulow asi- nasjszybsza wersja
"ASI_Prosty_Zapis"	FC 83	FC 83	// Prosty zapis danych do modulow Asi (nastawiony na predkosc)
"Opoznienie_Wylotu"	FC 85	FC 85
"FC_Bledy_KB1"	FC 117	FC 117
"FC_Bledy_KB2"	FC 118	FC 118
"FC_Bledy_Buff"	FC 119	FC 119
"FC_HMI_KB1"	FC 121	FC 121
"FC_HMI_KB2"	FC 122	FC 122
"FC_HMI_BUFF"	FC 123	FC 123
"FC_HMI_WOZEK"	FC 128	FC 128
"Funkcja_Zegara"	FC 140	FC 140	// Funkcja zegara
"Shuttle_Comand"	FC 200	FC 200
"Wymiana_Pakietow_Wozek"	FC 201	FC 201	// Wymiana duzej ilosci danych z wozkiem
"Komunikacja_Gender"	FC 205	FC 205
"Monitor_Bandy"	FC 313	FC 313	// Funkcja monitorujaca przejezdzajacy produkt
"Monitor_Bandy_2"	FC 314	FC 314	// Monitor Bandy z wykryciem auto
"Monitor_Bandy_+_Reczny"	FC 315	FC 315	// Funkcja monitorujaca + tryb reczny
"Monitor_Palety"	FC 316	FC 316	// Auto wyszukiwanie palety w masce
"Znajdz_Widmo"	FC 317	FC 317	// Funkcja szuka palety widmo
"Dekoduj_Maske"	FC 320	FC 320
"Dobor_Elementow_Lini"	FC 400	FC 400
"Opis_Dwubajtu_Zadanego"	FC 401	FC 401
"Sorting_FC"	FC 402	FC 402
"Shuttle_Queue"	FC 403	FC 403
"Wozek_Queue_V2"	FC 404	FC 404
"Sorting_V2"	FC 405	FC 405
"Wozek_Queue_V3"	FC 408	FC 408
"Sorting_V3"	FC 409	FC 409
"FC_Nawigator"	FC 410	FC 410
"Wozek_Jezdny_Kolejka"	FC 600	FC 600
"Send_Data"	FC 700	FC 700
"Receive_Data"	FC 701	FC 701
"Read_Data"	FC 702	FC 702
"Share_Data"	FC 703	FC 703	// Funkcja udostepniajaca dane
"Ekran_Para_Wozek"	FC 1701	FC 1701
"Ekran_Kier_KB1"	FC 1720	FC 1720
"Ekran_Kier_Rot"	FC 1721	FC 1721
"Ekran_Para_Odbieranie"	FC 1730	FC 1730
"PB_Strefa"	I 4.0	BOOL
"PB_Funkcja"	I 4.3	BOOL
"Obrtonica_Tyl"	I 5.1	BOOL
"Buff_PB_Reset_Przek_Bezp"	I 8.0	BOOL
"Buff_PB_Semi_Auto"	I 8.1	BOOL
"Buff_PB_Auto"	I 8.2	BOOL
"i_Buff_PB_Zal_Wozka"	I 8.3	BOOL
"Buff_Foto_Wozek_Pob"	I 8.7	BOOL
"Buf_Przek_Bezp_Ok"	I 10.0	BOOL
"Buff_Przek_Shuttle_OK"	I 10.1	BOOL
"KB1_PB_Reset_Bezp"	I 12.0	BOOL	// Przycisk kasowanie strefy bezpieczenstwa
"KB1_PB_Semi_Auto"	I 12.1	BOOL	// Przycisk polautomatyki
"KB1_PB_Auto"	I 12.2	BOOL	// Przycisk Automatyki
"KB1_PB_Funkcja"	I 12.3	BOOL
"KB1_PB_Shuttle_Tyl"	I 12.4	BOOL	// Przycisk shuttle przod
"KB1_PB_Shuttle_Przod"	I 12.5	BOOL	// Przycisk shuttle tyl
"KB1_PB_Winda_Przod"	I 12.6	BOOL	// Przycisk winda przod
"KB1_PB_Winda_Tyl"	I 12.7	BOOL	// Przycisk winda tyl
"KB1_PB_Obrotnica_Przod"	I 13.0	BOOL
"KB1_PB_Obrotnica_Tyl"	I 13.1	BOOL
"KB1_PB_Band_Seg_Przod"	I 13.2	BOOL	// Banda Segbetr przod
"KB1_PB_Band_Seg_Tyl"	I 13.3	BOOL	// Banda Segbert tyl
"KB1_PB_WWylot_2_Przod"	I 13.4	BOOL
"KB1_PB_WWylot_2_Tyl"	I 13.5	BOOL
"KB1_Rez_I23.6"	I 13.6	BOOL
"KB1_Rez_I23.7"	I 13.7	BOOL
"KB1_P_Bezp_Ok"	I 14.0	BOOL	// Przekaznik bezpieczenstwa ok
"KB1_P_Bezp_Shuttle_Ok"	I 14.1	BOOL	// Przekanik bezpieczenstwa Shuttle ok
"KB1_Petla_Fuse_Ok"	I 14.2	BOOL	// Petla bezpiecznikow Ok
"KB1_PB_Wyb_Obr_Lewo"	I 14.3	BOOL
"KB1_PB_Wyb_Obr_Prawo"	I 14.4	BOOL
"KB1_PB_Grzybek_Pracy"	I 14.5	BOOL
"KB1_PB_Pedal_Pracy_1"	I 14.6	BOOL
"KB1_PB_Pedal_Pracy_2"	I 14.7	BOOL
"KB1_Winda_W_Dole"	I 15.0	BOOL
"KB1_Winda_W_Gorze"	I 15.1	BOOL
"KB1_Foto_Shuttle"	I 15.2	BOOL
"KB1_Obecn_Wozka_Wylot_2"	I 15.3	BOOL
"KB1_Rezerwa_I25.4"	I 15.4	BOOL
"KB1_Rezerwa_I25.5"	I 15.5	BOOL
"KB1_Rezerwa_I25.6"	I 15.6	BOOL
"KB1_Rezerwa_I25.7"	I 15.7	BOOL
"KB1_Foto_Seg_Przod"	I 16.0	BOOL
"KB1_Foto_Segbert_Tyl"	I 16.1	BOOL
"KB1_Zasilanie_Seg_Fal"	I 16.2	BOOL	// Falowniki sa zasilane
"KB1_Obr_Foto_2"	I 17.0	BOOL
"KB1_Obr_Foto_1"	I 17.1	BOOL
"KB2_PB_Reset_Bezp"	I 22.0	BOOL	// Przycisk kasowanie strefy bezpieczenstwa
"KB2_PB_Semi_Auto"	I 22.1	BOOL	// Przycisk polautomatyki
"KB2_PB_Auto"	I 22.2	BOOL	// Przycisk Automatyki
"KB2_PB_Funkcja"	I 22.3	BOOL
"KB2_PB_Shuttle_Tyl"	I 22.4	BOOL	// Przycisk shuttle przod
"KB2_PB_Shuttle_Przod"	I 22.5	BOOL	// Przycisk shuttle tyl
"KB2_PB_Winda_Przod"	I 22.6	BOOL	// Przycisk winda przod
"KB2_PB_Winda_Tyl"	I 22.7	BOOL	// Przycisk winda tyl
"KB2_PB_Obrotnica_Przod"	I 23.0	BOOL
"KB2_PB_Obrotnica_Tyl"	I 23.1	BOOL
"KB2_PB_Band_Seg_Przod"	I 23.2	BOOL	// Banda Segbetr przod
"KB2_PB_Band_Seg_Tyl"	I 23.3	BOOL	// Banda Segbert tyl
"KB2_PB_WWylot_2_Przod"	I 23.4	BOOL
"KB2_PB_WWylot_2_Tyl"	I 23.5	BOOL
"KB2_Rez_I23.6"	I 23.6	BOOL
"KB2_Rez_I23.7"	I 23.7	BOOL
"KB2_P_Bezp_Ok"	I 24.0	BOOL	// Przekaznik bezpieczenstwa ok
"KB2_P_Bezp_Shuttle_Ok"	I 24.1	BOOL	// Przekanik bezpieczenstwa Shuttle ok
"KB2_Petla_Fuse_Ok"	I 24.2	BOOL	// Petla bezpiecznikow Ok
"KB2_PB_Wyb_Obr_Lewo"	I 24.3	BOOL
"KB2_PB_Wyb_Obr_Prawo"	I 24.4	BOOL
"KB2_PB_Grzybek_Pracy"	I 24.5	BOOL
"KB2_PB_Pedal_Pracy_1"	I 24.6	BOOL
"KB2_PB_Pedal_Pracy_2"	I 24.7	BOOL
"KB2_Winda_W_Dole"	I 25.0	BOOL
"KB2_Winda_W_Gorze"	I 25.1	BOOL
"KB2_Foto_Shuttle"	I 25.2	BOOL
"KB2_Obecn_Wozka_Wylot_2"	I 25.3	BOOL
"KB2_Rezerwa_I25.4"	I 25.4	BOOL
"KB2_Rezerwa_I25.5"	I 25.5	BOOL
"KB2_Rezerwa_I25.6"	I 25.6	BOOL
"KB2_Rezerwa_I25.7"	I 25.7	BOOL
"KB2_Foto_Seg_Przod"	I 26.0	BOOL
"KB2_Foto_Banda_Seg_Tyl"	I 26.1	BOOL
"KB2_Zasilanie_Seg_Fal"	I 26.2	BOOL
"KB2_Obr_Foto_2"	I 27.0	BOOL
"KB2_Obr_Foto_1"	I 27.1	BOOL
"ip_Bit_Kom_Shuttle"	I 30.0	BOOL	// bit komunikacji ( Shuttle <---)
"ip_Potw_Nowej_Pozycji"	I 31.1	BOOL	// Bit potwierdzenia przyjecia nowej pozycji (Shuttle <---)
"ip_Shuttle_Na_Pozycji"	I 31.2	BOOL	// Wozek na pozycji (Shuttle <--)
"ip_Shuttle_Stoi"	I 31.3	BOOL	// Wozek nie jedzie (Shuttle <--)
"ip_Potw_Zasprz"	I 31.4	BOOL	// Potwierdzenie zasprzeglenia (Shuttle <--)
"ip_Potw_Rozprz"	I 31.5	BOOL	// Potwierdzenie Rozprzeglenia (Shuttle <--)
"ip_Foto_Przod"	I 31.6	BOOL	// Fotokomorka wozek przod (Shuttle <--)
"ip_Foto_Wozek_Tyl"	I 31.7	BOOL	// Fotokomorka wozek tyl (Shuttle <--)
"Buff_2_PB_Reset_Przek_B"	I 80.0	BOOL
"Buff_2_PB_Semi_Auto"	I 80.1	BOOL
"Buff_2_PB_Auto"	I 80.2	BOOL
"Buff_2_PB_Banda_7_Lewo"	I 81.0	BOOL
"Buff_2_PB_Banda_7_Prawo"	I 81.1	BOOL
"Buff_2_PB_Banda_8_Lewo"	I 81.2	BOOL
"Buff_2_PB_Banda_8_Prawo"	I 81.3	BOOL
"Buff_2_PB_Banda_17_Lewo"	I 81.4	BOOL
"Buff_2_PB_Banda_17_Prawo"	I 81.5	BOOL
"Buff_2_PB_Banda_18_Lewo"	I 81.6	BOOL
"Buff_2_PB_Banda_18_Prawo"	I 81.7	BOOL
"Buff_2_PB_Banda_W_Lewo"	I 82.0	BOOL
"Buff_2_PB_Banda_W_Prawo"	I 82.1	BOOL
"Buff_2_Foto_Wlot_2"	I 82.2	BOOL
"Buff_2_Foto_Wlot_3"	I 82.3	BOOL
"Dword_0_Shuttle"	ID 30	DWORD
"ip_Poz_Akt_Wozka"	ID 34	DINT	// Pozycja aktualna wozka (Shuttle <--)
"Zawsze_True"	M 0.0	BOOL
"Zawsze_False"	M 0.1	BOOL
"Marka_X"	M 0.3	BOOL	// Marka output wszystko jedno
"Help_Start"	M 1.0	BOOL
"Help_Zbocze_Start"	M 1.1	BOOL
"Help_Start_2"	M 1.2	BOOL
"Marka_Bezpieczenstwa_0"	M 2.0	BOOL	// Marka_Bezpieczenstwa poziomu 0
"Marka_Start_Stop"	M 2.1	BOOL
"Marka_Bezpieczenstwa_2"	M 2.2	BOOL
"Rejon_Bindownicy_Stop"	M 2.3	BOOL
"Strefa_Bind_Ok"	M 2.4	BOOL
"Help_PB_Stop"	M 2.5	BOOL
"Edge_2_6"	M 2.6	BOOL
"Freeze"	M 2.7	BOOL
"Brak_Bledu"	M 3.0	BOOL
"Falowniki_OK"	M 3.1	BOOL
"Fuse_OK"	M 3.2	BOOL
"Help_Freeze"	M 3.3	BOOL
"Marka_Bezpieczenstwa_3"	M 3.4	BOOL
"Zezwolenie_Na_Wjazd"	M 3.5	BOOL	// Do stawiania lini
"Stop_Hmi"	M 3.7	BOOL
"Jedz_Na_Nowa_Pozycje"	M 20.0	BOOL
"Pozycja_Shuttle_Zadana"	M 20.1	BOOL
"Brak_Komunikacji_Shuttle"	M 20.2	BOOL
"Shuttle_Na_Pozycji"	M 20.3	BOOL	// Shuttle jest na pozycji zadanej
"Pozycja_Gorna_Ok"	M 20.4	BOOL
"Pozycja_Dolna_Ok"	M 20.5	BOOL
"Reset zadania"	M 20.6	BOOL
"Edge_M20.7"	M 20.7	BOOL
"Zasprzegnij_Wozek"	M 21.0	BOOL
"Rozprzeglenie_Wozka"	M 21.1	BOOL
"Wozek_zasprzeglony"	M 21.2	BOOL
"Pom_Bit_Zasprzeg"	M 21.4	BOOL
"Foto_Wozek_Przod"	M 22.0	BOOL	// Fotokomorka wozek przod
"Foto_Wozek_Tyl"	M 22.1	BOOL	// Fotokomorka wozek tyl
"Silnik_Banda_Wozek_lewo"	M 22.2	BOOL
"Silnik_Banda_Wozke_Prawo"	M 22.3	BOOL
"Foto_Wozek_Przod_Opoz"	M 22.4	BOOL
"Foto_Wozek_Tyl_Opoz"	M 22.5	BOOL
"Bezpieczne_Pokrycie_Foto"	M 22.6	BOOL
"Zasprzeglenie_KB1"	M 23.0	BOOL	// Wozek zasprzeglony do KB1
"Zasprzeglenie_KB2"	M 23.1	BOOL	// Wozek zasprzeglony do KB2
"Zasprzeglenie_Pob_I1"	M 23.2	BOOL	// Zasprzeglenie Intro pobieranie
"Zasprzeglenie_Gender"	M 23.3	BOOL	// Wozek zasprzeglony do Gender
"Zasprzeglenie_Odbieranie"	M 23.4	BOOL	// Wozek zasprzeglony do odbierania
"Banda_Wozka_Pracuje"	M 23.5	BOOL
"Zasprzeglenie_Pob_I2"	M 23.6	BOOL
"Zasprzeglenie_Pob_I3"	M 23.7	BOOL
"Wozek_Marka_Bezp"	M 24.0	BOOL	// Marka Bezpieczenstwa wozek
"Wozek_Odwrocone_Sygnaly"	M 24.1	BOOL
"Wozek_Auto_Reczny"	M 24.2	BOOL	// Auto reczny wozek
"Wozek_Zez_Od_Nastepnej"	M 24.3	BOOL
"Wozek_Dost_Od_Nast"	M 24.4	BOOL	// Paleta dostarczona sygnal od nastepnej
"Wozek_Zabierz_Od_Pop"	M 24.5	BOOL	// Sygnal zabierz od poprzedniej
"Wozek_Zez_Reczny_Od_Pop"	M 24.6	BOOL	// Sygnal zezwolenia recznego od poprzedniej
"Wozek_Przycisk_Tyl"	M 24.7	BOOL
"Wozek_Przycisk_Przod"	M 25.0	BOOL
"Bit_Resetu_Interfejsu"	M 25.1	BOOL
"Wozek_Reczny_Od_Nast"	M 25.2	BOOL
"Wozek_Zabierz_Do_Nast"	M 26.0	BOOL	// Sygnal wozka zabierz do nastepnej
"Wozek_Zez_Do_Pop"	M 26.1	BOOL
"Wozek_Paleta_Dost_Do_Pop"	M 26.2	BOOL	// Paleta dostarczona do poprzedniej
"Wozek_Zez_Reczny_Do_Nast"	M 26.3	BOOL
"Wozek_Zez_Reczny_Do_Pop"	M 26.4	BOOL
"Wozek_Nieb_Zajetosc"	M 26.5	BOOL
"Help_Widmo"	M 27.0	BOOL
"Foto_Woz_Odbieranie"	M 27.1	BOOL	// Foto woz na odbieraniu
"Na_Pozycji_KB1"	M 40.0	BOOL
"Na_Pozycji_KB2"	M 40.1	BOOL
"Na_Pozycji_Gender"	M 40.2	BOOL
"Na_Pozycji_Odbieranie"	M 40.3	BOOL
"Na_Pozycji_Pob_I1"	M 40.4	BOOL
"Na_Pozycji_Pob_I2"	M 40.5	BOOL
"Na_Pozycji_Pob_I3"	M 40.6	BOOL
"Jedz_Na_KB1"	M 50.0	BOOL
"Jedz_Na_KB2"	M 50.1	BOOL
"Jedz_Na_Gender"	M 50.2	BOOL
"Jedz_Na_Odbior"	M 50.3	BOOL
"Jedz_Na_Pob_I1"	M 50.4	BOOL
"Jedz_Na_Zadana"	M 50.5	BOOL
"Marka_Jazdy_Na_Nowa_Poz"	M 50.6	BOOL
"Edge_50.7"	M 50.7	BOOL
"Edge_M51.0"	M 51.0	BOOL
"Blokada_Pobierania_I1"	M 51.1	BOOL
"Jedz_Na_Pob_I2"	M 52.0	BOOL
"Jedz_Na_Pob_I3"	M 52.1	BOOL
"Edge_M53.0"	M 53.0	BOOL
"Blokada_Pobierania_I2"	M 53.1	BOOL
"Edge_M54.0"	M 54.0	BOOL
"Blokada_Pobierania_I3"	M 54.1	BOOL
"KB1_M_Bezpieczenstwa_0"	M 102.0	BOOL
"KB1_Auto_Reczny"	M 104.0	BOOL
"M106.0"	M 106.0	BOOL
"M106.1"	M 106.1	BOOL
"Zbocz_M106.2"	M 106.2	BOOL
"Zbocze_M106.3"	M 106.3	BOOL
"Warunek_Pustych_Kolbusow"	M 106.4	BOOL
"Zbocze_M106.5"	M 106.5	BOOL
"Paleta_Na_Pob_I1"	M 106.6	BOOL
"Blokuj_Pobieranie"	M 106.7	BOOL
"Edge_M107.0"	M 107.0	BOOL
"Edge_M107.1"	M 107.1	BOOL
"KB1_Tryb_Uzbr_Aktyw"	M 108.0	BOOL
"KB1_Bit_Ham_Sew"	M 110.0	BOOL
"KB1_Zez_Hand_Do_Nast"	M 110.1	BOOL
"KB1_M_Foto_Segbert"	M 111.0	BOOL
"KB1_Zab_od_Segbert"	M 111.1	BOOL
"KB1_B_Seg_Hand_Przod"	M 111.3	BOOL
"KB1_B_Seg_Auto_Przod"	M 111.4	BOOL
"KB1_Zezwolenie_Dla_Windy"	M 111.6	BOOL
"KB1_Warunki_Windy"	M 114.0	BOOL
"KB1_Warunki_Obrotnicy"	M 114.1	BOOL
"Edge_M114.2"	M 114.2	BOOL
"KB1_Wrunk_Przyjzd_Wozka"	M 114.3	BOOL
"KB1_Podwojny_Wlot"	M 120.0	BOOL	// 1-tak,0-nie
"KB1_Inline"	M 120.1	BOOL	// 1-tak,0-nie
"KB1_Uzbrajanie_Seg"	M 120.2	BOOL	// 1-tak,0-nie
"KB1_Uzbrajenie_Feedera"	M 120.3	BOOL	// 1-tak,0-nie
"KB1_Res_220_0_4"	M 120.4	BOOL
"KB1_Res_220_0_5"	M 120.5	BOOL
"KB1_Res_220_0_6"	M 120.6	BOOL
"KB1_Res_220_0_7"	M 120.7	BOOL
"KB1_VPB_Obrotnica_Przod"	M 121.0	BOOL	// VPB-virtual push button
"KB1_VPB_Obrotnica_Tyl"	M 121.1	BOOL	// VPB-virtual push button
"KB1_VPB_Obrotnica_CW"	M 121.2	BOOL	// VPB-virtual push button
"KB1_VPB_Obrotnica_CCW"	M 121.3	BOOL	// VPB-virtula push button
"KB1_Virutal_Foto_Wylot"	M 121.4	BOOL
"KB1_M121.5"	M 121.5	BOOL
"KB1_VPB_Winda_Przod"	M 122.0	BOOL
"KB1_VPB_Winda_Tyl"	M 122.1	BOOL
"KB1_VPB_Winda_Gora"	M 122.2	BOOL
"KB1_VPB_Winda_Dol"	M 122.3	BOOL
"KB1_Winda_Jazda_Gora"	M 122.4	BOOL
"KB1_Winda_Jazda_Dol"	M 122.5	BOOL
"KB1_Not_Aus_Pulpit_OK"	M 123.0	BOOL	// Not Aus adres 20 ok
"KB1_Grzyb_Bezp_OK"	M 123.1	BOOL	// Grzyb bezpieczenistwa Adres 21 OK
"KB1_Przek_Bezp_Potw"	M 123.3	BOOL	// Przekaznik bezpieczenstwa mozliwy do potwierdzenia
"KB1_Blada_Lini"	M 123.4	BOOL
"KB1_Uzbr_Oczek_Akt"	M 124.0	BOOL
"KB1_Start_Uzbr_Shot"	M 124.1	BOOL	// Krotki sygnal startu uzbrajania
"KB1_Sygnal_Kon_Uzbr"	M 124.2	BOOL	// Sygnal konca uzbrajania
"KB1_Pedal_W_Lewo"	M 124.3	BOOL	// Pedal obrotnicy jw lewo
"KB1_Pedal_W_Prawo"	M 124.4	BOOL	// Pedal obrotnicy jw prawo
"KB1_Uzbr_Aktywne"	M 124.5	BOOL	// Uzbrajanie palety jest aktywne
"KB1_Zez_Na_Uzbrajanie"	M 124.6	BOOL
"KB1_Uzbrj_Reczne"	M 124.7	BOOL
"KB1_Sygnal_Dzwiekowy"	M 125.0	BOOL
"KB1_Zbocze_M125.1"	M 125.1	BOOL
"KB1_Zez_Na_Uzbraj"	M 142.6	BOOL
"KB1_Help_Poz_1"	M 200.0	BOOL
"KB2_Help_Poz_1"	M 200.1	BOOL
"KB2_Help_Poz_2"	M 200.2	BOOL
"Buffory_Help_Poz_1"	M 200.3	BOOL
"Gender_Help_Poz_1"	M 200.4	BOOL
"Gender_Help_Poz_2"	M 200.5	BOOL
"KB2_M_Bezpieczenstwa_0"	M 202.0	BOOL
"KB2_Auto_Reczny"	M 204.0	BOOL	// 1-Auto,0-Reczny
"Edge_M207.0"	M 207.0	BOOL
"Edge_M207.1"	M 207.1	BOOL
"KB2_Tryb_Uzbr_Aktyw"	M 208.0	BOOL
"KB2_Bit_Ham_Sew"	M 210.0	BOOL
"KB2_Zez_Hand_Do_Nast"	M 210.1	BOOL
"KB2_M_Foto_Segbert"	M 211.0	BOOL
"KB2_Zab_od_Segbert"	M 211.1	BOOL
"KB2_B_Seg_Hand_Przod"	M 211.3	BOOL
"KB2_B_Seg_Auto_Przod"	M 211.4	BOOL
"KB2_Zezwolenie_Dla_Windy"	M 211.6	BOOL
"KB2_Warunki_Windy"	M 214.0	BOOL
"KB2_Warunki_Obrotnicy"	M 214.1	BOOL
"Edge_M214.2"	M 214.2	BOOL
"KB2_Wrunk_Przyjzd_Wozka"	M 214.3	BOOL
"KB2_Podwojny_Wlot"	M 220.0	BOOL	// 1-tak,0-nie
"KB2_Inline"	M 220.1	BOOL	// 1-tak,0-nie
"KB2_Uzbrajanie_Seg"	M 220.2	BOOL	// 1-tak,0-nie
"KB2_Uzbrajenie_Feedera"	M 220.3	BOOL	// 1-tak,0-nie
"KB2_Res_220_0_4"	M 220.4	BOOL
"KB2_Res_220_0_5"	M 220.5	BOOL
"KB2_Res_220_0_6"	M 220.6	BOOL
"KB2_Res_220_0_7"	M 220.7	BOOL
"KB2_VPB_Obrotnica_Przod"	M 221.0	BOOL	// VPB-virtual push button
"KB2_VPB_Obrotnica_Tyl"	M 221.1	BOOL	// VPB-virtual push button
"KB2_VPB_Obrotnica_CW"	M 221.2	BOOL	// VPB-virtual push button
"KB2_VPB_Obrotnica_CCW"	M 221.3	BOOL	// VPB-virtula push button
"KB2_Virutal_Foto_Wylot"	M 221.4	BOOL
"KB2_M221.5"	M 221.5	BOOL
"KB2_VPB_Winda_Przod"	M 222.0	BOOL
"KB2_VPB_Winda_Tyl"	M 222.1	BOOL
"KB2_VPB_Winda_Gora"	M 222.2	BOOL
"KB2_VPB_Winda_Dol"	M 222.3	BOOL
"KB2_Winda_Jazda_Gora"	M 222.4	BOOL
"KB2_Winda_Jazda_Dol"	M 222.5	BOOL
"KB2_Not_Aus_Pulpit_OK"	M 223.0	BOOL	// Not Aus adres 20 ok
"KB2_Grzyb_Bezp_OK"	M 223.1	BOOL	// Grzyb bezpieczenistwa Adres 21 OK
"KB2_Przek_Bezp_Potw"	M 223.3	BOOL	// Przekaznik bezpieczenstwa mozliwy do potwierdzenia
"KB2_Blada_Lini"	M 223.4	BOOL
"KB2_Uzbr_Oczek_Akt"	M 224.0	BOOL
"KB2_Start_Uzbr_Shot"	M 224.1	BOOL	// Krotki sygnal startu uzbrajania
"KB2_Sygnal_Kon_Uzbr"	M 224.2	BOOL	// Sygnal konca uzbrajania
"KB2_Pedal_W_Lewo"	M 224.3	BOOL	// Pedal obrotnicy jw lewo
"KB2_Pedal_W_Prawo"	M 224.4	BOOL	// Pedal obrotnicy jw prawo
"KB2_Uzbr_Aktywne"	M 224.5	BOOL	// Uzbrajanie palety jest aktywne
"KB2_Zez_Na_Uzbrajanie"	M 224.6	BOOL
"KB2_Uzbrj_Reczne"	M 224.7	BOOL
"KB2_Sygnal_Dzwiekowy"	M 225.0	BOOL
"KB2_Zbocze_M225.1"	M 225.1	BOOL
"Marka_Bezp_Buf_Prawe"	M 302.0	BOOL
"Silniki_Prawe_Ok"	M 302.3	BOOL
"Help_M302.7"	M 302.7	BOOL
"Marka_Bezp_Buf_Lewe"	M 303.0	BOOL
"Silniki_Lewe_Ok"	M 303.3	BOOL
"I1_Buf_Auto_Reczny"	M 304.0	BOOL
"I1_Buff_Opoz_Startu"	M 304.2	BOOL
"I2_Buff_Opoz_Startu"	M 304.3	BOOL
"I3_Buff_Opoz_Startu"	M 304.4	BOOL
"I2_I3_Buf_Auto_Reczny"	M 305.0	BOOL
"Buff_Obwody_Got_Do_Potw"	M 306.0	BOOL
"Edge_M307.0"	M 307.0	BOOL
"Edge_M307.1"	M 307.1	BOOL
"Edge_M308.0"	M 308.0	BOOL
"Edge_M308.1"	M 308.1	BOOL
"M_Miganie_200ms"	M 310.0	BOOL
"M_Miganie_500ms"	M 310.1	BOOL
"M_Miganie_100ms"	M 310.2	BOOL
"I1_Kier_Pob_Spedycja"	M 311.0	BOOL
"I1_Kier_Pob_Intro"	M 311.1	BOOL
"I1_Buff_Wiaz_Pop"	M 311.2	BOOL
"I1_Buff_Wiaz_Wzdl"	M 311.3	BOOL
"Blokuj_Czerwone"	M 312.0	BOOL
"Buff_Opoz_Foto_Wylot"	M 313.0	BOOL
"Help_M313.1"	M 313.1	BOOL
"Buff_Odbier_Wolne"	M 314.0	BOOL	// Miejsce na buforach jest wolne
"I1_Buff_Kod_0"	M 315.0	BOOL
"I1_Buff_Kod_1"	M 315.1	BOOL
"I1_Buff_Kod_2"	M 315.2	BOOL
"I1_Buff_Kod_3"	M 315.3	BOOL
"Stanowisko_I1"	M 315.4	BOOL
"I1_Stan_Ma_Zadanie"	M 315.5	BOOL
"Edge_M315.6"	M 315.6	BOOL
"Help_M315.7"	M 315.7	BOOL
"I2_Kier_Pob_Spedycja"	M 317.0	BOOL
"I2_Kier_Pob_Intro"	M 317.1	BOOL
"I2_Buff_Wiaz_Pop"	M 317.2	BOOL
"I2_Buff_Wiaz_Wzdl"	M 317.3	BOOL
"I2_Buff_Kod_0"	M 318.0	BOOL
"I2_Buff_Kod_1"	M 318.1	BOOL
"I2_Buff_Kod_2"	M 318.2	BOOL
"I2_Buff_Kod_3"	M 318.3	BOOL
"Stanowisko_I2"	M 318.4	BOOL
"I2_Stan_Ma_Zadanie"	M 318.5	BOOL
"Edge_M318.6"	M 318.6	BOOL
"Help_318.7"	M 318.7	BOOL
"I3_Kier_Pob_Spedycja"	M 319.0	BOOL
"I3_Kier_Pob_Intro"	M 319.1	BOOL
"I3_Buff_Wiaz_Pop"	M 319.2	BOOL
"I3_Buff_Wiaz_Wzdl"	M 319.3	BOOL
"I3_Buff_Kod_0"	M 320.0	BOOL
"I3_Buff_Kod_1"	M 320.1	BOOL
"I3_Buff_Kod_2"	M 320.2	BOOL
"I3_Buff_Kod_3"	M 320.3	BOOL
"Stanowisko_I3"	M 320.4	BOOL
"I3_Stan_Ma_Zadanie"	M 320.5	BOOL
"Edge_M320.6"	M 320.6	BOOL
"Help_320.7"	M 320.7	BOOL
"Brak_komunikacj_Gender"	M 400.0	BOOL
"Wspolny_Auto"	M 401.0	BOOL
"Wspolny_Reczny"	M 401.1	BOOL
"Zbocze_M401.2"	M 401.2	BOOL
"Gender_Zalacz_Auto_Woz"	M 401.7	BOOL	// Gender ma zalaczyc auto wozkowi
"Gender_Auto_Reczny"	M 404.0	BOOL
"Reset_Read"	M 501.0	BOOL	// Przycisk resetu transmisji
"Toggle_Para"	M 501.1	BOOL
"BL_Read_K_KB1"	M 502.0	BOOL
"Bl_Na_Write_K_KB1"	M 502.1	BOOL
"Help_Timmer_KB"	M 502.2	BOOL
"Help_M502.3"	M 502.3	BOOL
"Kier_KB1_Koniec_Read"	M 502.5	BOOL
"Kier_KB1_Koniec_Send"	M 502.6	BOOL
"Aktywna_Funkcja_KB"	M 502.7	BOOL
"Bl_Na_Read_K_Rot"	M 503.0	BOOL
"Bl_Na_Write_K_Rot"	M 503.1	BOOL
"Help_Timmer_Rot"	M 503.2	BOOL
"Help_M503.3"	M 503.3	BOOL
"Kier_Rot_Koniec_Read"	M 503.5	BOOL
"Kier_Rot_Koniec_Send"	M 503.6	BOOL
"Aktywna_Funkcja_Rot"	M 503.7	BOOL
"Bl_Na_Read_Para"	M 504.0	BOOL
"Bl_Na_Write_Para"	M 504.1	BOOL
"Help_Timmer_Para"	M 504.2	BOOL
"Help_M504.3"	M 504.3	BOOL
"Para_Koniec_Read"	M 504.5	BOOL
"Para_Koniec_Send"	M 504.6	BOOL
"Aktywna_Funkcja_Para"	M 504.7	BOOL
"Bl_Na_Read_Odb"	M 505.0	BOOL
"Bl_Na_Write_Odb"	M 505.1	BOOL
"Help_Timmer_Odb"	M 505.2	BOOL
"Help_M505.3"	M 505.3	BOOL
"Odb_Koniec_Read"	M 505.5	BOOL
"Odb_Koniec_Send"	M 505.6	BOOL
"Aktywna_Funkcja_Odb"	M 505.7	BOOL
"Edge_M513.0"	M 513.0	BOOL
"Edge_M513.1"	M 513.1	BOOL
"Edge_513.4"	M 513.4	BOOL
"Edge_M513.5"	M 513.5	BOOL
"Edge_M514.0"	M 514.0	BOOL
"M514.1"	M 514.1	BOOL
"Edge_M514.3"	M 514.3	BOOL
"Edge_M514.4"	M 514.4	BOOL
"Edge_M523.0"	M 523.0	BOOL
"Edge_M523.1"	M 523.1	BOOL
"Edge_M533.0"	M 533.0	BOOL
"Edge_M533.1"	M 533.1	BOOL
"Paleta_Obecna_Na_KB1"	M 600.0	BOOL
"Paleta_Obecna_Na_KB2"	M 600.1	BOOL
"Paleta_Obecna_Pob_I1"	M 600.3	BOOL
"Paleta_Obecna_Pob_I2"	M 600.4	BOOL
"Paleta_Obecna_Pob_I3"	M 600.5	BOOL
"Foto_Pokryte_Czasowo"	M 600.6	BOOL
"Foto_Odkryte_Czasowo"	M 600.7	BOOL
"Wpisz_Wartosc_Do_Stosu"	M 601.0	BOOL
"Kasuj_Rekord_W_Kolejce"	M 601.1	BOOL
"Pobierz_Wartosc"	M 601.2	BOOL
"Potwierdzenie_Wpisania"	M 602.0	BOOL
"Potwierdzenie_Pobrania"	M 602.1	BOOL
"Potwierdzenie_Kasowania"	M 602.2	BOOL
"Help_M602.3"	M 602.3	BOOL
"Help_M602.4"	M 602.4	BOOL
"Help_M602.5"	M 602.5	BOOL
"Przejmij_Z_KB1"	M 603.0	BOOL
"Przejmij_Z_KB2"	M 603.1	BOOL
"Przejmij_Z_I1"	M 603.2	BOOL
"Oddaj_Na_Spedycje"	M 603.3	BOOL
"Oddaj_Na_Intro"	M 603.4	BOOL
"Przejmij_z_I2"	M 603.5	BOOL
"Przejmij_z_I3"	M 603.6	BOOL
"Wozek_Na_Reczny"	M 605.0	BOOL
"Wozek_Na_Auto"	M 605.1	BOOL
"Edge_M606.0"	M 606.0	BOOL
"Edge_M606.1"	M 606.1	BOOL
"Edge_M606.2"	M 606.2	BOOL
"Edge_M606.3"	M 606.3	BOOL
"KB1_Przej_Auto_Na_Recz"	M 607.0	BOOL
"KB2_Przej_Auto_Na_Recz"	M 607.1	BOOL
"Buff_Przejscie_Na_Recz"	M 607.2	BOOL
"Gen_Przejscie_Na_Reczny"	M 607.3	BOOL
"Edge_M608.0"	M 608.0	BOOL
"Edge_M608.1"	M 608.1	BOOL
"Edge_M608.2"	M 608.2	BOOL
"Edge_M608.3"	M 608.3	BOOL
"Warunk_Zasprz_KB1"	M 609.0	BOOL
"Warunk_Zasprz_KB2"	M 609.1	BOOL
"Warunk_Zasprz_Buffory"	M 609.2	BOOL
"Warunk_Zasprz_Gender"	M 609.3	BOOL
"Wozek_Kier_Spedycja"	M 610.0	BOOL
"Wozek_Kier_Intro"	M 610.1	BOOL
"Wozek_Info_Bit_0"	M 611.0	BOOL
"Wozek_Info_Bit_1"	M 611.1	BOOL
"Wozek_Info_Bit_2"	M 611.2	BOOL
"Wozek_Info_Bit_3"	M 611.3	BOOL
"Edge_M612.0"	M 612.0	BOOL
"Help_M612.1"	M 612.1	BOOL
"Paleta_Od_KB12"	M 615.0	BOOL
"Pozcja_Wozek_Zadana"	MD 10	DINT
"Offset_Pozycji"	MD 14	DINT
"Gorny_Zakres_Pozycji_Ok"	MD 28	DINT
"Dolny_Zakres_Pozycji_Ok"	MD 32	DINT
"KB1_MD140"	MD 140	DINT
"KB1_Cale_Zadanie"	MD 148	DWORD
"KB2_MD240"	MD 240	DINT
"KB2_Cale_Zadanie"	MD 248	DINT
"Help_MD340"	MD 340	DINT
"I1_Buff_Mask_Dword"	MD 360	DWORD
"I2_Buff_Mask_Dword"	MD 380	DWORD
"Help_MD382"	MD 382	DINT
"Help_MD384"	MD 384	DINT
"I3_Buff_Mask_Dword"	MD 390	DWORD
"I3_Help_MD394"	MD 394	DINT
"Wartosc_Dla_Wozka"	MD 620	DINT
"Wartosc_Wyjsciowa_Sortu"	MD 624	DINT
"Help_MD628"	MD 628	DWORD
"Kod_Przejdu_Do_Wozka"	MD 634	DINT
"War_KB1_Waga"	MD 650	DINT
"War_KB2_Waga"	MD 654	DINT
"War_I1_Waga"	MD 658	DINT
"War_I2_Waga"	MD 662	DINT
"War_I3_Waga"	MD 666	DINT
"Rejestr_Wozka"	MD 680	DWORD
"Wartosc_Bufforu_Help"	MD 720	DWORD
"KB1_Rozkaz_Zadania"	MW 148	WORD
"Wartosc_Bufforu_W_Kol"	MW 160	INT
"KB2_Rozkaz_Zadania"	MW 248	WORD
"Help_MW350"	MW 350	WORD
"Help_MW352"	MW 352	WORD
"Help_MW354"	MW 354	WORD
"Help_Mw356"	MW 356	WORD
"Help_MW358"	MW 358	WORD
"I1_Buff_Maska_Z_HMI"	MW 360	WORD
"Help_MW370"	MW 370	WORD
"Help_MW372"	MW 372	WORD
"Help_MW374"	MW 374	WORD
"Help_MW376"	MW 376	WORD
"Help_MW378"	MW 378	WORD
"I2_Buff_Maska_Z_HMI"	MW 380	WORD
"I3_Buff_Maska_Z_HMI"	MW 390	WORD
"I2_Help_MW412"	MW 412	WORD
"I2_Help_MW414"	MW 414	WORD
"I3_Help_MW416"	MW 416	WORD
"I3_Help_MW418"	MW 418	WORD
"Help_MW520"	MW 520	WORD
"Help_MW522"	MW 522	WORD
"Petla_Read_Kier_KB1"	MW 524	INT
"Petla_Send_Kier_KB1"	MW 526	INT
"MW530"	MW 530	WORD
"Help_MW532"	MW 532	WORD
"Petla_Read_Kier_Rot"	MW 534	INT
"Petla_Send_Kier_Rot"	MW 536	INT
"Help_MW540"	MW 540	WORD
"Help_MW542"	MW 542	WORD
"Petla_Read_Para"	MW 544	INT
"Petla_Send_Para"	MW 546	INT
"Help_MW628"	MW 628	WORD
"MW_Kolejka_KB1"	MW 670	INT
"MW_Kolejka_KB2"	MW 672	INT
"MW_Kolejka_I1"	MW 674	INT
"MW_Kolejka_I2"	MW 676	INT
"MW_Kolejka_I3"	MW 678	INT
"I/O_FLT1"	OB 82	OB 82	// I/O Point Fault 1
"RACK_FLT"	OB 86	OB 86	// Loss of Rack Fault
"COMM_FLT"	OB 87	OB 87	// Communication Fault
"PROG_ERR"	OB 121	OB 121	// Programming Error
"MOD_ERR"	OB 122	OB 122	// Module Access Error
"Buff_Lam_Przek_Bezp_O"	Q 8.0	BOOL	// Przekaznik bezpieczenstwa buffory ok
"Buff_Lampka_Pol_Auto"	Q 8.1	BOOL
"Buffor_Lampka_Auto"	Q 8.2	BOOL
"q_Buff_Zal_Wozka"	Q 8.3	BOOL
"q_Reset_P_Bezp_KB1"	Q 8.4	BOOL	// Reset przekaznika bezpieczenstwa Wozka KB1 s.18
"q_Reset_P_Bezp_KB2"	Q 8.5	BOOL	// Reset przekaznika bezpieczenstwa Wozka KB2 s.18
"Rezerwa_Q8.6"	Q 8.6	BOOL
"Rezerwa_Q8.7"	Q 8.7	BOOL
"Rezerwa_Q9.0"	Q 9.0	BOOL
"Rezerwa_Q9.1"	Q 9.1	BOOL
"Buff_Lampa_Kol_Buf_Ziel"	Q 9.2	BOOL
"Buff_Lampa_Kol_Buf_Pom"	Q 9.3	BOOL
"Buff_Lampa_Kol_Buf_Czer"	Q 9.4	BOOL
"Buff_Lampa_Kol_Buf_Nieb"	Q 9.5	BOOL
"Buff_Lampa_Kol_Buf_Syg"	Q 9.6	BOOL
"Rezerwa_Q9.7"	Q 9.7	BOOL
"Buff_Reset_Przek_Bezp"	Q 10.0	BOOL
"Buff_Reset_Przek_Bezp_1"	Q 10.1	BOOL
"Buff_Reset_Przeka_Bezp_2"	Q 10.2	BOOL
"Buff_Swiatlo_Zielone"	Q 10.3	BOOL	// Swiatlo zielone drogowe
"Buff_Swiatl_Czerwone"	Q 10.4	BOOL
"Rezerwa_Q10.5"	Q 10.5	BOOL
"Rezerwa_Q10.6"	Q 10.6	BOOL
"Rezerwa_Q10.7"	Q 10.7	BOOL
"Buff_Lampa_Kol_Gen_Ziel"	Q 11.0	BOOL	// S
"Buff_Lampa_Kol_Gen_Pom"	Q 11.1	BOOL	// str 21
"Buff_Lampa_Kol_Gen_Czer"	Q 11.2	BOOL	// str 21
"Buff_Lampa_Kol_Gen_Bial"	Q 11.3	BOOL	// str 21
"Buff_Lampa_Kol_Gen_Syg"	Q 11.4	BOOL	// str 21
"Rezerwa_Q11.6"	Q 11.5	BOOL	// str 21
"KB1_PB_Strefa_B_Lampka"	Q 12.0	BOOL	// Lapmka strefa bezpieczenstwa ok
"KB1_PB_Semi_Auto_Lampka"	Q 12.1	BOOL	// Lampka polautomatyka
"KB1_PB_Auto_Lampka"	Q 12.2	BOOL	// Lampka auto
"KB1_PB_Funkcja_Lampka"	Q 12.3	BOOL	// Lampka przycisku funkcyjnego
"KB1_PB_B_Winda_Lampka"	Q 12.4	BOOL	// Lampka piorka winda
"KB1_PB_B_Obr_Lampka"	Q 12.5	BOOL	// Lampka piorka obrotnica
"KB1_Rezerwa_Q22.6"	Q 12.6	BOOL
"KB1_Rezerwa_Q22.7"	Q 12.7	BOOL
"KB1_Lampa_Wyb_Kier_Lewo"	Q 13.0	BOOL
"KB1_Lampa_Wyb_Kier_Prawo"	Q 13.1	BOOL
"KB1_Lampa_Kol_Ziel"	Q 13.2	BOOL	// Lampka kolor zielony str 19
"KB1_Lampa_Kol_Pom"	Q 13.3	BOOL	// Lampka kolor pomaranczowy str 19
"KB1_Lampa_Kol_Czerw"	Q 13.4	BOOL	// Lampka kolor czerwony str 19
"KB1_Lampa_Kol_Nieb"	Q 13.5	BOOL
"KB1_Syrena"	Q 13.6	BOOL
"KB1_Lampa_Blysk_Wozek"	Q 13.7	BOOL
"KB1_Winda_Silnik_Pompa"	Q 14.0	BOOL
"KB1_Winda_Zawor"	Q 14.1	BOOL
"KB1_Reset_Przek_Bezp"	Q 14.2	BOOL
"KB1_Odblokuj_Lenze"	Q 14.3	BOOL
"KB1_Przek_Rez_K20.5"	Q 14.4	BOOL
"KB1_Odblokuj_Ham_Sew"	Q 14.5	BOOL
"KB1_Odblokuj_Ham_Lenze"	Q 14.6	BOOL
"KB1_Rezerwa_Q24.7"	Q 14.7	BOOL
"KB1_Fal_Seg_Przod"	Q 15.0	BOOL
"KB1_Fal_Segbert_Tyl"	Q 15.1	BOOL
"KB2_PB_Strefa_B_Lampka"	Q 22.0	BOOL	// Lapmka strefa bezpieczenstwa ok
"KB2_PB_Semi_Auto_Lampka"	Q 22.1	BOOL	// Lampka polautomatyka
"KB2_PB_Auto_Lampka"	Q 22.2	BOOL	// Lampka auto
"KB2_PB_Funkcja_Lampka"	Q 22.3	BOOL	// Lampka przycisku funkcyjnego
"KB2_PB_B_Winda_Lampka"	Q 22.4	BOOL	// Lampka piorka winda
"KB2_PB_B_Obr_Lampka"	Q 22.5	BOOL	// Lampka piorka obrotnica
"KB2_Rezerwa_Q22.6"	Q 22.6	BOOL
"KB2_Rezerwa_Q22.7"	Q 22.7	BOOL
"KB2_Lampa_Wyb_Kier_Lewo"	Q 23.0	BOOL
"KB2_Lampa_Wyb_Kier_Prawo"	Q 23.1	BOOL
"KB2_Lampa_Kol_Ziel"	Q 23.2	BOOL	// Lampka kolor zielony str 19
"KB2_Lampa_Kol_Pom"	Q 23.3	BOOL	// Lampka kolor pomaranczowy str 19
"KB2_Lampa_Kol_Czerw"	Q 23.4	BOOL	// Lampka kolor czerwony str 19
"KB2_Lampa_Kol_Nieb"	Q 23.5	BOOL
"KB2_Syrena"	Q 23.6	BOOL
"KB2_Lampa_Blysk_Wozek"	Q 23.7	BOOL
"KB2_Winda_Silnik_Pompa"	Q 24.0	BOOL
"KB2_Winda_Zawor"	Q 24.1	BOOL
"KB2_Reset_Przek_Bezp"	Q 24.2	BOOL
"KB2_Odblokuj_Lenze"	Q 24.3	BOOL
"KB2_Przek_Rez_K20.5"	Q 24.4	BOOL
"KB2_Odblokuj_Ham_Sew"	Q 24.5	BOOL
"KB2_Odblokuj_Ham_Lenze"	Q 24.6	BOOL
"KB2_Rezerwa_Q24.7"	Q 24.7	BOOL
"KB2_Fal_Seg_Przod"	Q 25.0	BOOL
"KB2_Fal_Seg_Tyl"	Q 25.1	BOOL
"op_Bit_Komunikacji"	Q 38.0	BOOL	// Bit komunikacji do Shuttle(-->Shuttle)
"op_Bit_Nowej_Pozycji"	Q 39.1	BOOL	// Bit zadania nowej pozycji (-->Shuttle)
"op_Potw_Pozycji"	Q 39.2	BOOL	// Bit potwierdzenia pzosycji (-->Shuttle)
"op_Bit_Rezerwy_38_3"	Q 39.3	BOOL	// Bit rezerwy 38.3
"op_Zasprz_Wozka"	Q 39.4	BOOL	// Rozkaz Zasprzeglenie Wozka (-->Shuttle)
"op_Rozprz_Wozka"	Q 39.5	BOOL	// Rozkaz Rozprzeglenie Wozka (--> Shuttle)
"op_Silnik_Banda_Lewo"	Q 39.6	BOOL	// Jazda silnika w lewo (-->Shuttle)
"op_Silnik_Banda_Prawo"	Q 39.7	BOOL	// Jazda silnika w prawo
"Buff_1_Wlot_1_Wiaz_Pop"	Q 80.0	BOOL
"Buff_1_Wlot_1_Wiaz_Wzdl"	Q 80.1	BOOL
"Buff_1_Wlot_1_Dekl"	Q 80.2	BOOL
"Buff_1_Wlot_1_Fol"	Q 80.3	BOOL
"Buff_2_Wlot_2_Wiaz_Pop"	Q 80.4	BOOL
"Buff_2_Wlot_2_Wiaz_Wzdl"	Q 80.5	BOOL
"Buff_2_Wlot_2_Dekl"	Q 80.6	BOOL
"Buff_2_Wlot_2_Fol"	Q 80.7	BOOL
"Buff_2_Wlot_3_Wiaz_Pop"	Q 81.0	BOOL
"Buff_2_Wlot_3_Wiaz_Wzdl"	Q 81.1	BOOL
"Buff_2_Wlot_3_Dekl"	Q 81.2	BOOL
"Buff_2_Wlot_3_Fol"	Q 81.3	BOOL
"Buff_2_Lampka_Strefa_B"	Q 82.0	BOOL
"Buff_2_Lampka_Pol_Auto"	Q 82.1	BOOL
"Buff_2_Lampka_Auto"	Q 82.2	BOOL
"DWORD_8_Shuttle"	QD 38	DWORD
"QD42_Pozycja_Zadana"	QD 42	DINT	// Pozycja zadana w mm (--> Shuttle)
"READ_CLK"	SFC 1	SFC 1	// Read System Clock
"DPNRM_DG"	SFC 13	SFC 13	// Read Diagnostic Data of a DP Slave
"DPRD_DAT"	SFC 14	SFC 14	// Read Consistent Data of a Standard DP Slave
"DPWR_DAT"	SFC 15	SFC 15	// Write Consistent Data to a Standard DP Slave
"BLKMOV"	SFC 20	SFC 20	// Copy Variables
"READ_ERR"	SFC 38	SFC 38	// Read Error Registers
"WR_REC"	SFC 58	SFC 58	// Write Data Record
"RD_REC"	SFC 59	SFC 59	// Read a Data Record
"Timer_0_Czerwone"	T 0	TIMER
"Timer_T1"	T 1	TIMER
"Shuttle_T2"	T 2	TIMER
"Help_T4"	T 4	TIMER
"KB1_T10"	T 10	TIMER
"KB1_T11"	T 11	TIMER
"KB1_T12"	T 12	TIMER
"KB1_T13"	T 13	TIMER
"KB1_T14"	T 14	TIMER
"KB1_T15"	T 15	TIMER
"KB1_Opoznienie_Startu"	T 16	TIMER
"KB1_Filtr_Segbert"	T 17	TIMER
"KB1_T18"	T 18	TIMER
"T19"	T 19	TIMER
"KB2_T20"	T 20	TIMER
"KB2_T21"	T 21	TIMER
"KB2_T22"	T 22	TIMER
"KB2_T23"	T 23	TIMER
"KB2_T24"	T 24	TIMER
"KB2_T25"	T 25	TIMER
"KB2_Opoznienie_Startu"	T 26	TIMER
"KB2_Filtr_Segbert"	T 27	TIMER
"KB2_T28"	T 28	TIMER
"T29"	T 29	TIMER
"200ms_T31"	T 31	TIMER
"500ms_T32"	T 32	TIMER
"100ms_T33"	T 33	TIMER
"Buff_T35"	T 35	TIMER
"Buff_T36"	T 36	TIMER
"Buff_T37"	T 37	TIMER
"Kontrola_T40"	T 40	TIMER
"Kontrola_T41"	T 41	TIMER
"Kontrola_T42"	T 42	TIMER
"Kontrola_T43"	T 43	TIMER
"Kontrola_T44"	T 44	TIMER
"Kontrola_T45"	T 45	TIMER
"Kontrola_T46"	T 46	TIMER
"Kontrola_T47"	T 47	TIMER
"Kontrola_T48"	T 48	TIMER
"Kontrola_T49"	T 49	TIMER
"KB1_T50"	T 50	TIMER
"KB1_T51"	T 51	TIMER
"KB1_T52"	T 52	TIMER
"Kontrola_T53"	T 53	TIMER
"Kontrola_T54"	T 54	TIMER
"Kontrola_T55"	T 55	TIMER
"Kontrola_T56"	T 56	TIMER
"KB2_T60"	T 60	TIMER
"KB2_T61"	T 61	TIMER
"KB2_T62"	T 62	TIMER
"BUF_T70"	T 70	TIMER
"T71_Opoznienie_Rozp"	T 71	TIMER
"Timer_Wozek_Pokryte"	T 72	TIMER
"Timer_Wozek_Odkryte"	T 73	TIMER
"T75"	T 75	TIMER
"T76"	T 76	TIMER
"T77"	T 77	TIMER
"T78"	T 78	TIMER
"T79"	T 79	TIMER
"Help_T80"	T 80	TIMER
"Help_T81"	T 81	TIMER
"Help_T82"	T 82	TIMER
"Help_T90"	T 90	TIMER
"KB2_Timer_Winda_91"	T 91	TIMER
"KB2_Timer_Winda_92"	T 92	TIMER
"KB1_Timer_Winda_93"	T 93	TIMER
"KB1_Timer_Winda_94"	T 94	TIMER
"T100"	T 100	TIMER
"T_100_Wozek_Na_Auto"	T 101	TIMER
"Timmer_102_KB1"	T 102	TIMER
"Timer_103_KB2"	T 103	TIMER
"Timmer_104_Pobieranie"	T 104	TIMER
"Timmer_105_Odbieranie"	T 105	TIMER
"Help_T107"	T 107	TIMER
"Help_T108"	T 108	TIMER
"T109"	T 109	TIMER
"Timmer_T110"	T 110	TIMER
"Timmer_T111"	T 111	TIMER
"Timmer_Pob_I2"	T 112	TIMER
"Timmer_Pob_I3"	T 113	TIMER
"Timer_T120"	T 120	TIMER
"Help_T121"	T 121	TIMER
"t122"	T 122	TIMER
"T130"	T 130	TIMER
"T131"	T 131	TIMER
"T140"	T 140	TIMER
"T141"	T 141	TIMER
"T150"	T 150	TIMER
"TASMA_MODEL"	UDT 1	UDT 1	// Model Tasmy z Sew'em
"ESTOP_MODEL"	UDT 3	UDT 3
"OBROTNICA_MODEL"	UDT 6	UDT 6	// Model sygnalow z bandy obrotowej
"CZUJNIKI_MODEL_1"	UDT 7	UDT 7	// Model czujnikow na obrotnicy
"VAT_1"	VAT 1	
"Wejscia_Wysjcia"	VAT 2	
"VAT_DB701"	VAT 3	
"VAT_DB702"	VAT 4	
"VAT_kb2"	VAT 5	
"para"	VAT 6	
"VAT_Buffory"	VAT 7	
"VAT_Cargo"	VAT 8	
"buffory_2"	VAT 9	
END_SYMBOL_TABLE

TYPE "TASMA_MODEL"	// UDT 1
VERSION : 0.1
  STRUCT
   Silnik_OK : BOOL ;	//Silnik ok
   Rezerwa_Silnik : BOOL ;
   Foto_1 : BOOL ;	//Wejscie SEW 1
   Foto_2 : BOOL ;	//Wejscie SEW 2
   C_Wise : BOOL ;	//ClockWise
   CC_Wise : BOOL ;	//CounterClockWise
   Wolno : BOOL ;	//Wolno
   S_Bit : BOOL ;	//Bit bezpieczenstwa
   Zez_Do_Pop : BOOL ;	//Zezwolenie do poprzedniej
   Paleta_Dost_do_Pop : BOOL ;	//Potwierdzenie dostarczenia
   Zabierz_do_Nast : BOOL ;	//Przejecie palety do nast
   Paleta_Poprawna : BOOL ;	//Wykorzystywane do monitoringu
   Paleta_Na_Stanowisku : BOOL ;	//Paleta obecna na stanowisku
   Res_1_5 : BOOL ;
   Zez_Reczny_do_Pop : BOOL ;	//Zezwolenie na reczny tyl
   Zez_Reczny_do_Nast : BOOL ;	//Zezwolenie na reczny przod
   Res_2_0 : BOOL ;
   Res_2_1 : BOOL ;
   Res_2_2 : BOOL ;
   Res_2_3 : BOOL ;
   Res_2_4 : BOOL ;
   Res_2_5 : BOOL ;
   Res_2_6 : BOOL ;
   Res_2_7 : BOOL ;
   Res_3_0 : BOOL ;
   Res_3_1 : BOOL ;
   Res_3_2 : BOOL ;
   Res_3_3 : BOOL ;
   Res_3_4 : BOOL ;
   Res_3_5 : BOOL ;
   Res_3_6 : BOOL ;
   Res_3_7 : BOOL ;
  END_STRUCT ;	
END_TYPE

TYPE "ESTOP_MODEL"	// UDT 3
VERSION : 0.1
  STRUCT
   EStop_Tor_1_1 : BOOL ;
   EStop_Tor_1_2 : BOOL ;
   EStop_Tor_2_1 : BOOL ;
   EStop_Tor_2_2 : BOOL ;
   Rez_0_4 : BOOL ;
   Rez_0_5 : BOOL ;
   Rez_0_6 : BOOL ;
   Rez_0_7 : BOOL ;
   Rez_1_0 : BOOL ;
   Rez_1_1 : BOOL ;
   Rez_1_2 : BOOL ;
   Rez_1_3 : BOOL ;
   Rez_1_4 : BOOL ;
   Rez_1_5 : BOOL ;
   Rez_1_6 : BOOL ;
   Rez_1_7 : BOOL ;
   Res_2_0 : BOOL ;
   Res_2_1 : BOOL ;
   Res_2_2 : BOOL ;
   Res_2_3 : BOOL ;
   Res_2_4 : BOOL ;
   Res_2_5 : BOOL ;
   Res_2_6 : BOOL ;
   Res_2_7 : BOOL ;
   Res_3_0 : BOOL ;
   Res_3_1 : BOOL ;
   Res_3_2 : BOOL ;
   Res_3_3 : BOOL ;
   Res_3_4 : BOOL ;
   Res_3_5 : BOOL ;
   Res_3_6 : BOOL ;
   Res_3_7 : BOOL ;
  END_STRUCT ;	
END_TYPE

TYPE "OBROTNICA_MODEL"	// UDT 6
VERSION : 0.1
  STRUCT
   Silnik_OK : BOOL ;	//Silnik ok
   Rezerwa_Silnik : BOOL ;
   Foto_1 : BOOL ;	//Wejscie SEW 1
   Foto_2 : BOOL ;	//Wejscie SEW 2
   C_Wise : BOOL ;	//ClockWise
   CC_Wise : BOOL ;	//CounterClockWise
   Wolno : BOOL ;	//Wolno
   S_Bit : BOOL ;	//Bit bezpieczenstwa
   Zez_Do_Pop_Wlot : BOOL ;	//Zezwolenie do poprzedniej
   Potw_Dost_Wlot : BOOL ;	//Potwierdzenie dostarczenia
   Zez_Do_Pop_Wlot_2 : BOOL ;	//Wykorzystywane do monitoringu
   Potw_Dost_Wlot_2 : BOOL ;
   Przejmij_Palete_Wylot_1 : BOOL ;	//Przejecie palety do nast
   Przejmij_Palete_Wylot_2 : BOOL ;
   Res_1_7 : BOOL ;
   Res_2_0 : BOOL ;
   Zezwolenie_Reczny_Pop : BOOL ;
   Zez_Reczny_Wylot_1 : BOOL ;
   Zez_Reczny_Wylot_2 : BOOL ;
   Res_2_4 : BOOL ;
   Res_2_5 : BOOL ;
   Res_2_6 : BOOL ;
   Res_2_7 : BOOL ;
   Res_3_0 : BOOL ;
   Res_3_1 : BOOL ;
   Res_3_2 : BOOL ;
   Res_3_3 : BOOL ;
   Res_3_4 : BOOL ;
   Res_3_5 : BOOL ;
   Res_3_6 : BOOL ;
   Res_3_7 : BOOL ;
  END_STRUCT ;	
END_TYPE

TYPE "CZUJNIKI_MODEL_1"	// UDT 7
VERSION : 0.1
  STRUCT
   Czujnik_0_St : BOOL ;
   Czujnik_Ham_0_St : BOOL ;
   Czujnik_Ham_90_St : BOOL ;
   Czujnik_90_St : BOOL ;
   Rez_0_4 : BOOL ;
   Rez_0_5 : BOOL ;
   Rez_0_6 : BOOL ;
   Rez_0_7 : BOOL ;
   Rez_1_0 : BOOL ;
   Rez_1_1 : BOOL ;
   Rez_1_2 : BOOL ;
   Rez_1_3 : BOOL ;
   Rez_1_4 : BOOL ;
   Rez_1_5 : BOOL ;
   Rez_1_6 : BOOL ;
   Rez_1_7 : BOOL ;
   Res_2_0 : BOOL ;
   Res_2_1 : BOOL ;
   Res_2_2 : BOOL ;
   Res_2_3 : BOOL ;
   Res_2_4 : BOOL ;
   Res_2_5 : BOOL ;
   Res_2_6 : BOOL ;
   Res_2_7 : BOOL ;
   Res_3_0 : BOOL ;
   Res_3_1 : BOOL ;
   Res_3_2 : BOOL ;
   Res_3_3 : BOOL ;
   Res_3_4 : BOOL ;
   Res_3_5 : BOOL ;
   Res_3_6 : BOOL ;
   Res_3_7 : BOOL ;
  END_STRUCT ;	
END_TYPE

FUNCTION_BLOCK "Stan_Shuttle"	// FB 1
//Funkcja sluzy do zlinkowania poszczegolnych stanowisk pracy z wozkiem jezdnym
AUTHOR : Kng
NAME : Main
VERSION : 0.1
VAR
  Shuttle_Band : FB 32;
END_VAR
BEGIN
NETWORK
TITLE =
//Ten Network celowo jest wolny
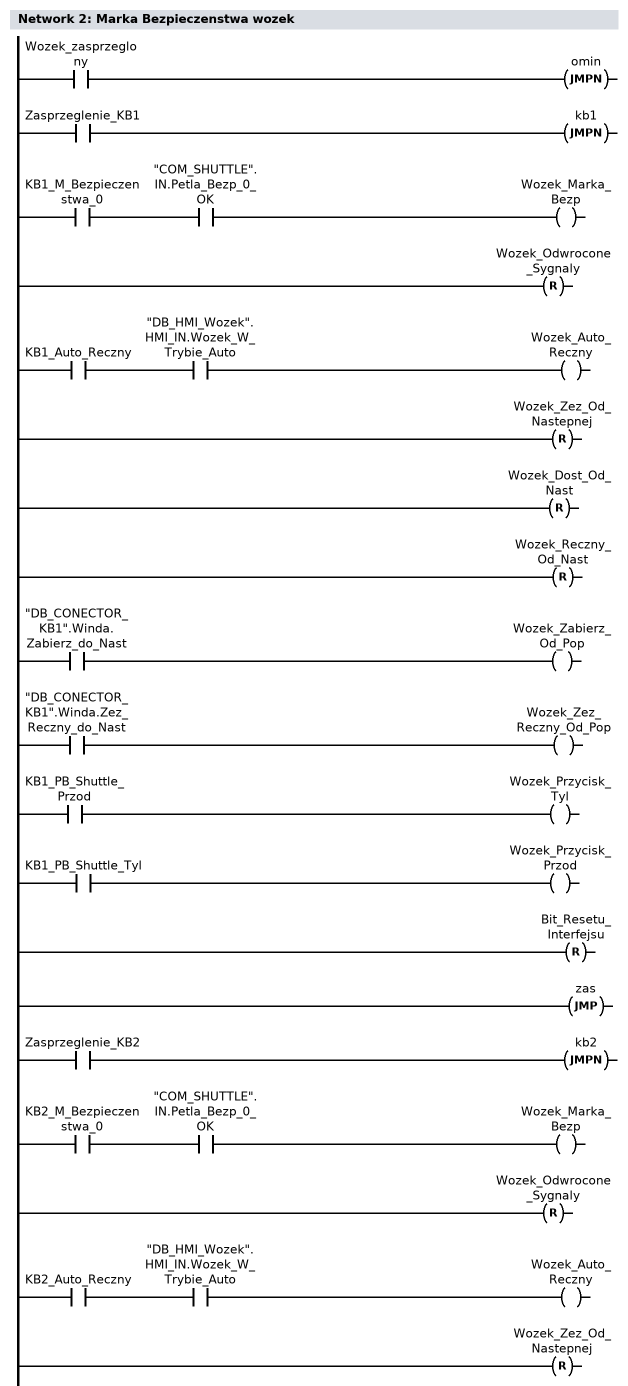
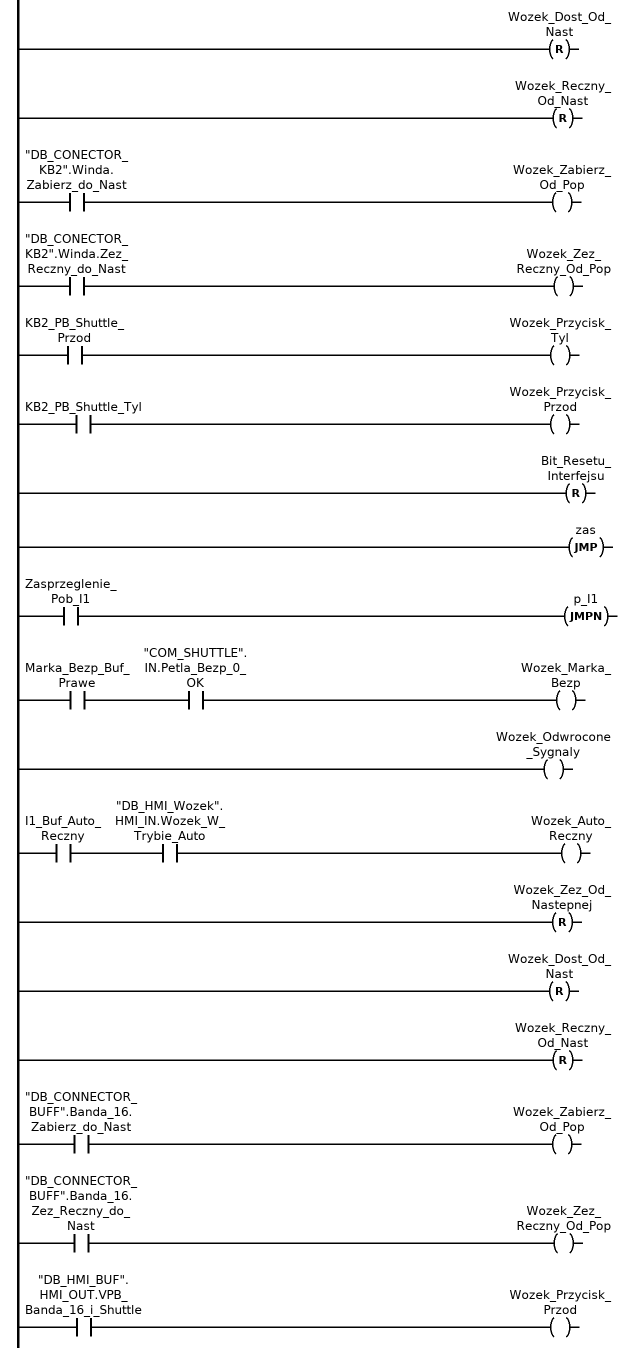
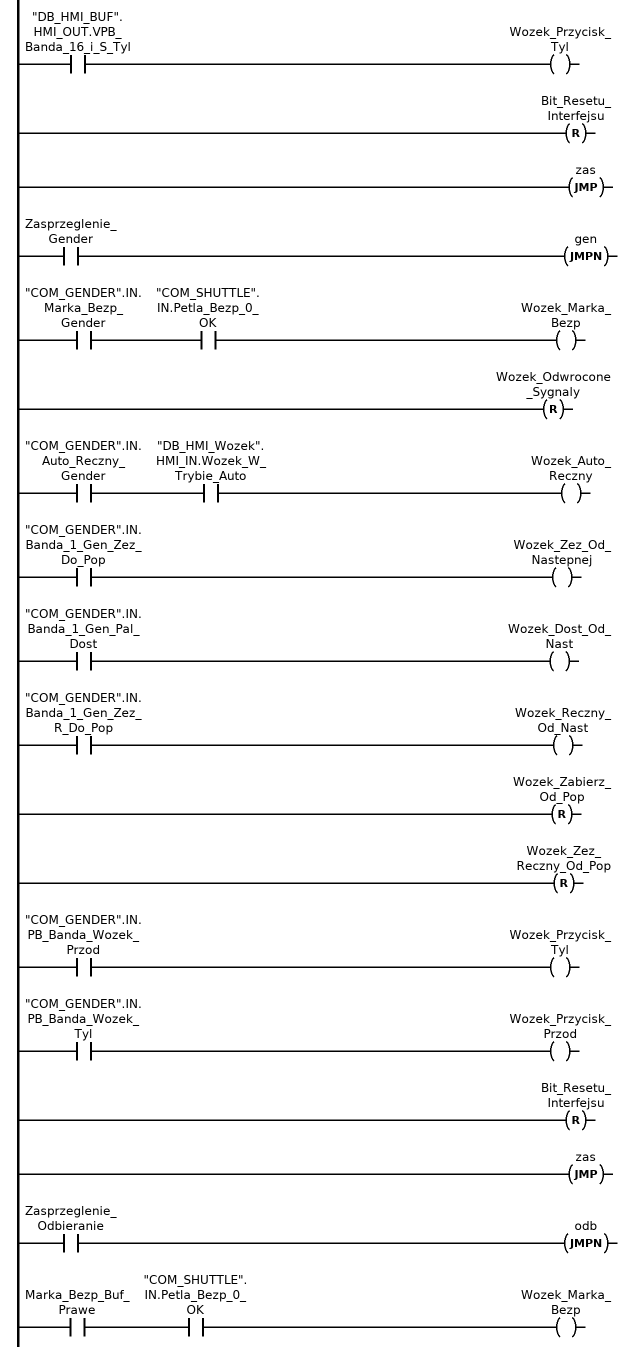
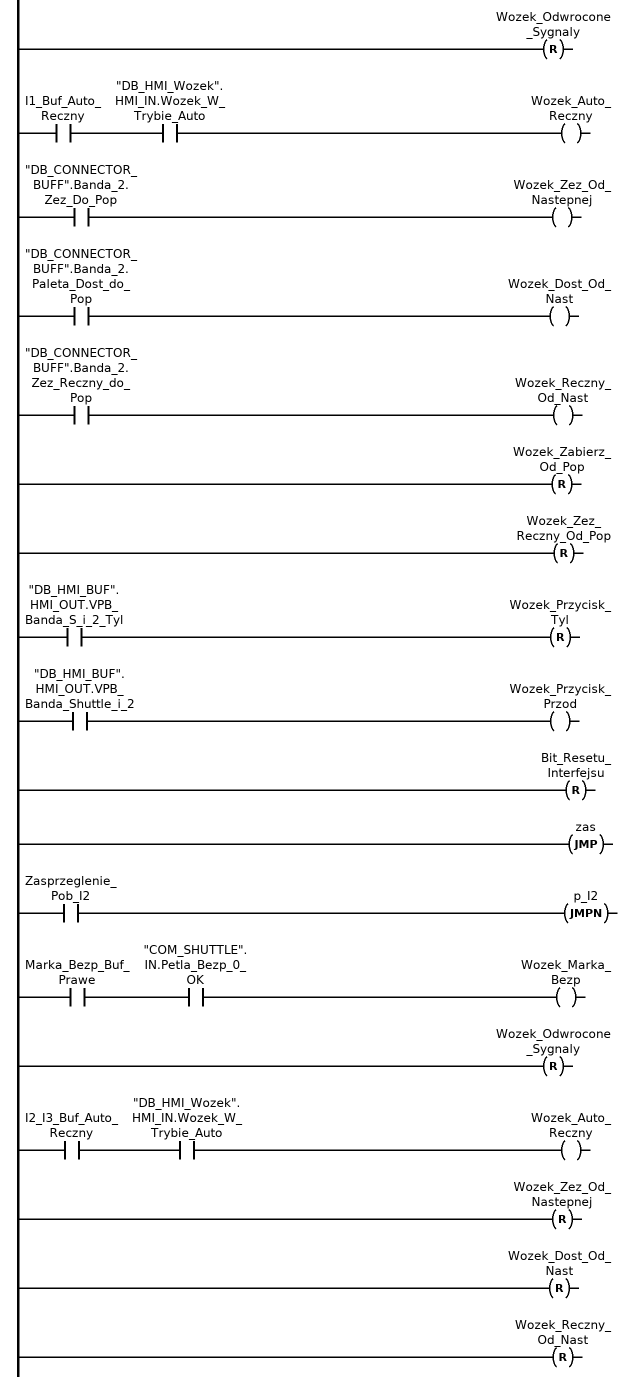
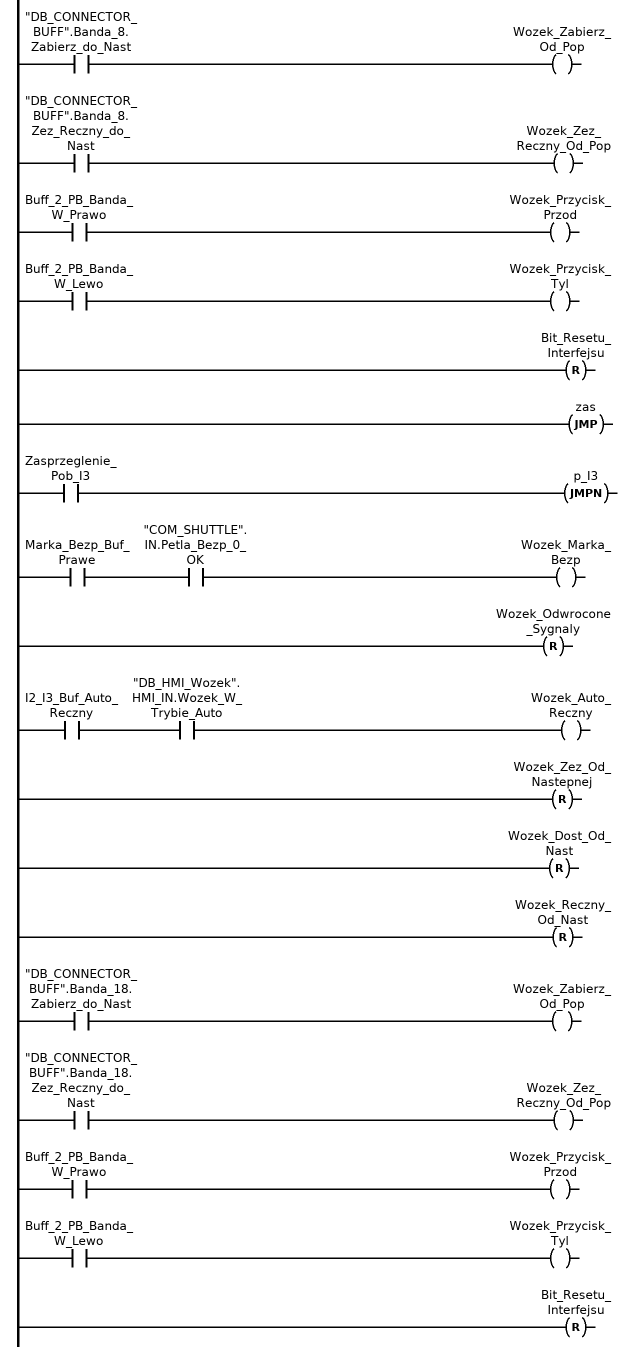
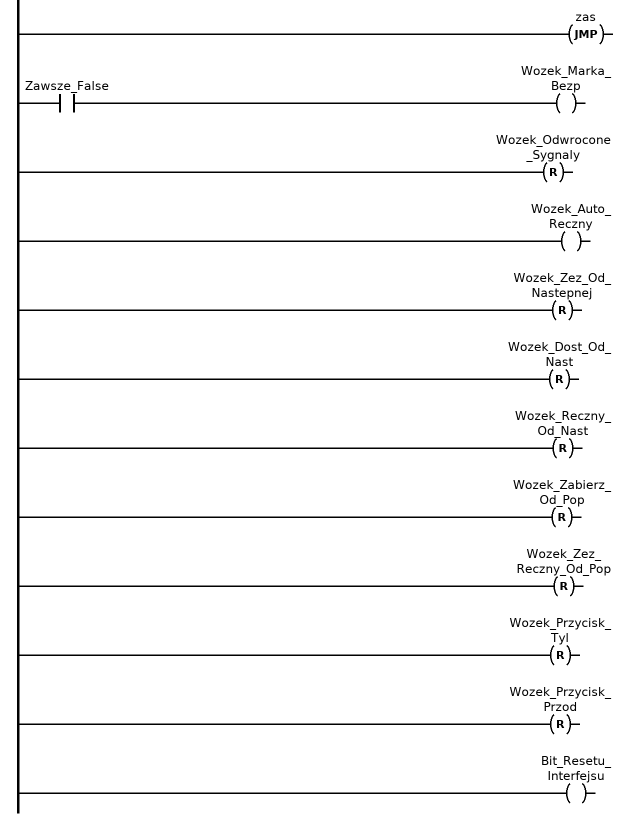
NETWORK
TITLE = Marka Bezpieczenstwa wozek
//Przepisanie bitow do bitow wejsciowych bandy (inputy)
      A     "Wozek_zasprzeglony";
      JCN   omin;
//******************KB1**********************************
      A     "Zasprzeglenie_KB1";
      JCN   kb1;
//***Marka bezpieczenstwa
      A     "KB1_M_Bezpieczenstwa_0";
      A     "COM_SHUTTLE".IN.Petla_Bezp_0_OK;
      =     "Wozek_Marka_Bezp";
//***Odwrocenie sygnalow
      SET;
      R     "Wozek_Odwrocone_Sygnaly";
//***Auto-reczny
      A     "KB1_Auto_Reczny";
      A     "DB_HMI_Wozek".HMI_IN.Wozek_W_Trybie_Auto;
      =     "Wozek_Auto_Reczny";
//***Zezwolenie od nastepnej
      SET;
      R     "Wozek_Zez_Od_Nastepnej";
//***Paleta dostarczona od nastepnej
      SET;
      R     "Wozek_Dost_Od_Nast";
//***Zezwolenie reczny od nastepnej
      SET;
      R     "Wozek_Reczny_Od_Nast";
//***Sygnal zabierz od poprzedniej
      A     "DB_CONECTOR_KB1".Winda.Zabierz_do_Nast;
      =     "Wozek_Zabierz_Od_Pop";
//***Zezwolenie reczny od poprzedniej
      A     "DB_CONECTOR_KB1".Winda.Zez_Reczny_do_Nast;
      =     "Wozek_Zez_Reczny_Od_Pop";
//***Przycisk recznej jazdy przod
      A     "KB1_PB_Shuttle_Przod";
      =     "Wozek_Przycisk_Tyl";
//***Przycisk recznej jazdy tyl
      A     "KB1_PB_Shuttle_Tyl";
      =     "Wozek_Przycisk_Przod";
//***Wejscier resetu interfejsu
      SET;
      R     "Bit_Resetu_Interfejsu";
//***skok bandy
      JU    zas;
kb1:  NOP   0;
//******************KB2*********************************
      A     "Zasprzeglenie_KB2";
      JCN   kb2;
//***Marka bezpieczenstwa
      A     "KB2_M_Bezpieczenstwa_0";
      A     "COM_SHUTTLE".IN.Petla_Bezp_0_OK;
      =     "Wozek_Marka_Bezp";
//***Odwrocenie sygnalow
      SET;
      R     "Wozek_Odwrocone_Sygnaly";
//***Auto-reczny
      A     "KB2_Auto_Reczny";
      A     "DB_HMI_Wozek".HMI_IN.Wozek_W_Trybie_Auto;
      =     "Wozek_Auto_Reczny";
//***Zezwolenie od nastepnej
      SET;
      R     "Wozek_Zez_Od_Nastepnej";
//***Paleta dostarczona od nastepnej
      SET;
      R     "Wozek_Dost_Od_Nast";
//***Zezwolenie reczny od nastepnej
      SET;
      R     "Wozek_Reczny_Od_Nast";
//***Sygnal zabierz od poprzedniej
      A     "DB_CONECTOR_KB2".Winda.Zabierz_do_Nast;
      =     "Wozek_Zabierz_Od_Pop";
//***Zezwolenie reczny od poprzedniej
      A     "DB_CONECTOR_KB2".Winda.Zez_Reczny_do_Nast;
      =     "Wozek_Zez_Reczny_Od_Pop";
//***Przycisk recznej jazdy przod
      A     "KB2_PB_Shuttle_Przod";
      =     "Wozek_Przycisk_Tyl";
//***Przycisk recznej jazdy tyl
      A     "KB2_PB_Shuttle_Tyl";
      =     "Wozek_Przycisk_Przod";
//***Wejscie resetu interfejsu
      SET;
      R     "Bit_Resetu_Interfejsu";
//***skok bandy
      JU    zas;
kb2:  NOP   0;
//******************Pobieranie I1 *********************************
      A     "Zasprzeglenie_Pob_I1";
      JCN   p_I1;
//***Marka bezpieczenstwa
      A     "Marka_Bezp_Buf_Prawe";
      A     "COM_SHUTTLE".IN.Petla_Bezp_0_OK;
      =     "Wozek_Marka_Bezp";
//***Odwrocenie sygnalow   !!!
      SET;
      =     "Wozek_Odwrocone_Sygnaly";
//***Auto-reczny
      A     "I1_Buf_Auto_Reczny";
      A     "DB_HMI_Wozek".HMI_IN.Wozek_W_Trybie_Auto;
      =     "Wozek_Auto_Reczny";
//***Zezwolenie od nastepnej
      SET;
      R     "Wozek_Zez_Od_Nastepnej";
//***Paleta dostarczona od nastepnej
      SET;
      R     "Wozek_Dost_Od_Nast";
//***Zezwolenie reczny od nastepnej
      SET;
      R     "Wozek_Reczny_Od_Nast";
//***Sygnal zabierz od poprzedniej
      A     "DB_CONNECTOR_BUFF".Banda_16.Zabierz_do_Nast;
      =     "Wozek_Zabierz_Od_Pop";
//***Zezwolenie reczny od poprzedniej
      A     "DB_CONNECTOR_BUFF".Banda_16.Zez_Reczny_do_Nast;
      =     "Wozek_Zez_Reczny_Od_Pop";
//***Przycisk recznej jazdy przod
      A     "DB_HMI_BUF".HMI_OUT.VPB_Banda_16_i_Shuttle;
      =     "Wozek_Przycisk_Przod";
//***Przycisk recznej jazdy tyl
      A     "DB_HMI_BUF".HMI_OUT.VPB_Banda_16_i_S_Tyl;
      =     "Wozek_Przycisk_Tyl";
//***Wejscie resetu interfejsu
      SET;
      R     "Bit_Resetu_Interfejsu";
//***skok bandy
      JU    zas;
p_I1: NOP   0;
//******************Gender*********************************
      A     "Zasprzeglenie_Gender";
      JCN   gen;
//***Marka bezpieczenstwa
      A     "COM_GENDER".IN.Marka_Bezp_Gender;
      A     "COM_SHUTTLE".IN.Petla_Bezp_0_OK;
      =     "Wozek_Marka_Bezp";
//***Odwrocenie sygnalow   
      SET;
      R     "Wozek_Odwrocone_Sygnaly";
//***Auto-reczny
      A     "COM_GENDER".IN.Auto_Reczny_Gender;
      A     "DB_HMI_Wozek".HMI_IN.Wozek_W_Trybie_Auto;
      =     "Wozek_Auto_Reczny";
//***Zezwolenie od nastepnej
      A     "COM_GENDER".IN.Banda_1_Gen_Zez_Do_Pop;
      =     "Wozek_Zez_Od_Nastepnej";
//***Paleta dostarczona od nastepnej
      A     "COM_GENDER".IN.Banda_1_Gen_Pal_Dost;
      =     "Wozek_Dost_Od_Nast";
//***Zezwolenie reczny od nastepnej
      A     "COM_GENDER".IN.Banda_1_Gen_Zez_R_Do_Pop;
      =     "Wozek_Reczny_Od_Nast";
//***Sygnal zabierz od poprzedniej
      SET;
      R     "Wozek_Zabierz_Od_Pop";
//***Zezwolenie reczny od poprzedniej
      SET;
      R     "Wozek_Zez_Reczny_Od_Pop";
//***Przycisk recznej jazdy przod
      A     "COM_GENDER".IN.PB_Banda_Wozek_Przod;
      =     "Wozek_Przycisk_Tyl";
//***Przycisk recznej jazdy tyl
      A     "COM_GENDER".IN.PB_Banda_Wozek_Tyl;
      =     "Wozek_Przycisk_Przod";
//***Wejscie resetu interfejsu
      SET;
      R     "Bit_Resetu_Interfejsu";
//***skok bandy
      JU    zas;
gen:  NOP   0;
//******************Odbieranie*********************************
      A     "Zasprzeglenie_Odbieranie";
      JCN   odb;
//***Marka bezpieczenstwa
      A     "Marka_Bezp_Buf_Prawe";
      A     "COM_SHUTTLE".IN.Petla_Bezp_0_OK;
      =     "Wozek_Marka_Bezp";
//***Odwrocenie sygnalow   
      SET;
      R     "Wozek_Odwrocone_Sygnaly";
//***Auto-reczny
      A     "I1_Buf_Auto_Reczny";
      A     "DB_HMI_Wozek".HMI_IN.Wozek_W_Trybie_Auto;
      =     "Wozek_Auto_Reczny";
//***Zezwolenie od nastepnej
      A     "DB_CONNECTOR_BUFF".Banda_2.Zez_Do_Pop;
      =     "Wozek_Zez_Od_Nastepnej";
//***Paleta dostarczona od nastepnej
      A     "DB_CONNECTOR_BUFF".Banda_2.Paleta_Dost_do_Pop;
      =     "Wozek_Dost_Od_Nast";
//***Zezwolenie reczny od nastepnej
      A     "DB_CONNECTOR_BUFF".Banda_2.Zez_Reczny_do_Pop;
      =     "Wozek_Reczny_Od_Nast";
//***Sygnal zabierz od poprzedniej
      SET;
      R     "Wozek_Zabierz_Od_Pop";
//***Zezwolenie reczny od poprzedniej
      SET;
      R     "Wozek_Zez_Reczny_Od_Pop";
//***Przycisk recznej jazdy przod
      A     "DB_HMI_BUF".HMI_OUT.VPB_Banda_S_i_2_Tyl;
      R     "Wozek_Przycisk_Tyl";
//***Przycisk recznej jazdy tyl
      A     "DB_HMI_BUF".HMI_OUT.VPB_Banda_Shuttle_i_2;
      =     "Wozek_Przycisk_Przod";
//***Wejscie resetu interfejsu
      SET;
      R     "Bit_Resetu_Interfejsu";
//***skok bandy
      JU    zas;
odb:  NOP   0;
//******************Pobieranie I2 *********************************
      A     "Zasprzeglenie_Pob_I2";
      JCN   p_I2;
//***Marka bezpieczenstwa
      A     "Marka_Bezp_Buf_Prawe";
      A     "COM_SHUTTLE".IN.Petla_Bezp_0_OK;
      =     "Wozek_Marka_Bezp";
//***Odwrocenie sygnalow   !!!
      SET;
      R     "Wozek_Odwrocone_Sygnaly";
//***Auto-reczny
      A     "I2_I3_Buf_Auto_Reczny";
      A     "DB_HMI_Wozek".HMI_IN.Wozek_W_Trybie_Auto;
      =     "Wozek_Auto_Reczny";
//***Zezwolenie od nastepnej
      SET;
      R     "Wozek_Zez_Od_Nastepnej";
//***Paleta dostarczona od nastepnej
      SET;
      R     "Wozek_Dost_Od_Nast";
//***Zezwolenie reczny od nastepnej
      SET;
      R     "Wozek_Reczny_Od_Nast";
//***Sygnal zabierz od poprzedniej
      A     "DB_CONNECTOR_BUFF".Banda_8.Zabierz_do_Nast;
      =     "Wozek_Zabierz_Od_Pop";
//***Zezwolenie reczny od poprzedniej
      A     "DB_CONNECTOR_BUFF".Banda_8.Zez_Reczny_do_Nast;
      =     "Wozek_Zez_Reczny_Od_Pop";
//***Przycisk recznej jazdy przod
      A     "Buff_2_PB_Banda_W_Prawo";
      =     "Wozek_Przycisk_Przod";
//***Przycisk recznej jazdy tyl
      A     "Buff_2_PB_Banda_W_Lewo";
      =     "Wozek_Przycisk_Tyl";
//***Wejscie resetu interfejsu
      SET;
      R     "Bit_Resetu_Interfejsu";
//***skok bandy
      JU    zas;
p_I2: NOP   0;
//******************Pobieranie I3 *********************************
      A     "Zasprzeglenie_Pob_I3";
      JCN   p_I3;
//***Marka bezpieczenstwa
      A     "Marka_Bezp_Buf_Prawe";
      A     "COM_SHUTTLE".IN.Petla_Bezp_0_OK;
      =     "Wozek_Marka_Bezp";
//***Odwrocenie sygnalow   !!!
      SET;
      R     "Wozek_Odwrocone_Sygnaly";
//***Auto-reczny
      A     "I2_I3_Buf_Auto_Reczny";
      A     "DB_HMI_Wozek".HMI_IN.Wozek_W_Trybie_Auto;
      =     "Wozek_Auto_Reczny";
//***Zezwolenie od nastepnej
      SET;
      R     "Wozek_Zez_Od_Nastepnej";
//***Paleta dostarczona od nastepnej
      SET;
      R     "Wozek_Dost_Od_Nast";
//***Zezwolenie reczny od nastepnej
      SET;
      R     "Wozek_Reczny_Od_Nast";
//***Sygnal zabierz od poprzedniej
      A     "DB_CONNECTOR_BUFF".Banda_18.Zabierz_do_Nast;
      =     "Wozek_Zabierz_Od_Pop";
//***Zezwolenie reczny od poprzedniej
      A     "DB_CONNECTOR_BUFF".Banda_18.Zez_Reczny_do_Nast;
      =     "Wozek_Zez_Reczny_Od_Pop";
//***Przycisk recznej jazdy przod
      A     "Buff_2_PB_Banda_W_Prawo";
      =     "Wozek_Przycisk_Przod";
//***Przycisk recznej jazdy tyl
      A     "Buff_2_PB_Banda_W_Lewo";
      =     "Wozek_Przycisk_Tyl";
//***Wejscie resetu interfejsu
      SET;
      R     "Bit_Resetu_Interfejsu";
//***skok bandy
      JU    zas;
p_I3: NOP   0;
omin: NOP   0;
//******************Wozek Rozprzeglony*********************************
//***Marka bezpieczenstwa
      A     "Zawsze_False";
      =     "Wozek_Marka_Bezp";
//***Odwrocenie sygnalow   
      SET;
      R     "Wozek_Odwrocone_Sygnaly";
//***Auto-reczny
      SET;
      =     "Wozek_Auto_Reczny";
//***Zezwolenie od nastepnej
      SET;
      R     "Wozek_Zez_Od_Nastepnej";
//***Paleta dostarczona od nastepnej
      SET;
      R     "Wozek_Dost_Od_Nast";
//***Zezwolenie reczny od nastepnej
      SET;
      R     "Wozek_Reczny_Od_Nast";
//***Sygnal zabierz od poprzedniej
      SET;
      R     "Wozek_Zabierz_Od_Pop";
//***Zezwolenie reczny od poprzedniej
      SET;
      R     "Wozek_Zez_Reczny_Od_Pop";
//***Przycisk recznej jazdy przod
      SET;
      R     "Wozek_Przycisk_Tyl";
//***Przycisk recznej jazdy tyl
      SET;
      R     "Wozek_Przycisk_Przod";
//***Wejscie resetu interfejsu
      SET;
      =     "Bit_Resetu_Interfejsu";
zas:  NOP   0;
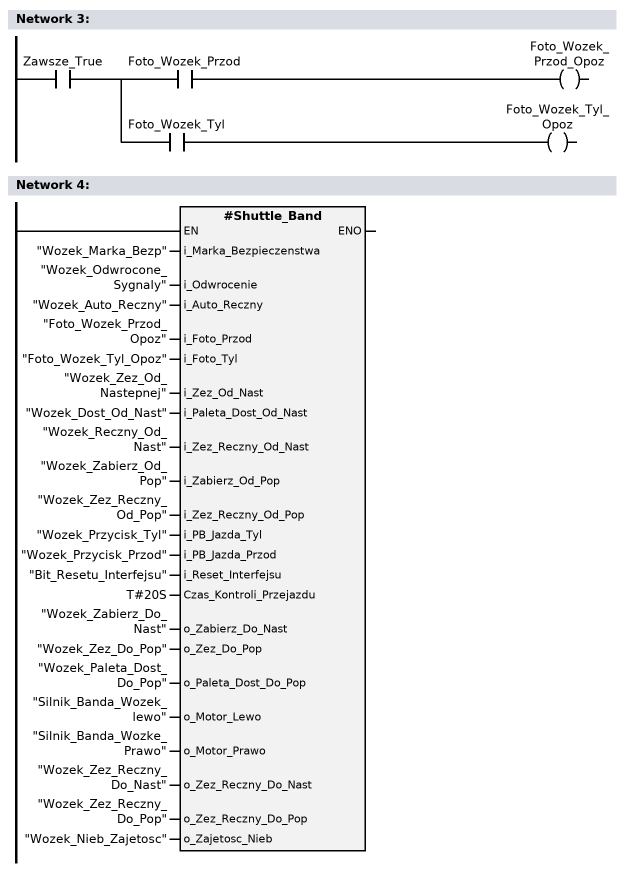
NETWORK
TITLE =
//Wydluzzenie czasow fotokomorek
      A     "Zawsze_True";
      =     L 0.0;
      A     L 0.0;
      A     "Foto_Wozek_Przod";
      =     "Foto_Wozek_Przod_Opoz";
      A     L 0.0;
      A     "Foto_Wozek_Tyl";
      =     "Foto_Wozek_Tyl_Opoz";
NETWORK
TITLE =
//Banda Wozek 
      CALL  #Shuttle_Band (
           i_Marka_Bezpieczenstwa   := "Wozek_Marka_Bezp",
           i_Odwrocenie             := "Wozek_Odwrocone_Sygnaly",
           i_Auto_Reczny            := "Wozek_Auto_Reczny",
           i_Foto_Przod             := "Foto_Wozek_Przod_Opoz",
           i_Foto_Tyl               := "Foto_Wozek_Tyl_Opoz",
           i_Zez_Od_Nast            := "Wozek_Zez_Od_Nastepnej",
           i_Paleta_Dost_Od_Nast    := "Wozek_Dost_Od_Nast",
           i_Zez_Reczny_Od_Nast     := "Wozek_Reczny_Od_Nast",
           i_Zabierz_Od_Pop         := "Wozek_Zabierz_Od_Pop",
           i_Zez_Reczny_Od_Pop      := "Wozek_Zez_Reczny_Od_Pop",
           i_PB_Jazda_Tyl           := "Wozek_Przycisk_Tyl",
           i_PB_Jazda_Przod         := "Wozek_Przycisk_Przod",
           i_Reset_Interfejsu       := "Bit_Resetu_Interfejsu",
           Czas_Kontroli_Przejazdu  := T#20S,
           o_Zabierz_Do_Nast        := "Wozek_Zabierz_Do_Nast",
           o_Zez_Do_Pop             := "Wozek_Zez_Do_Pop",
           o_Paleta_Dost_Do_Pop     := "Wozek_Paleta_Dost_Do_Pop",
           o_Motor_Lewo             := "Silnik_Banda_Wozek_lewo",
           o_Motor_Prawo            := "Silnik_Banda_Wozke_Prawo",
           o_Zez_Reczny_Do_Nast     := "Wozek_Zez_Reczny_Do_Nast",
           o_Zez_Reczny_Do_Pop      := "Wozek_Zez_Reczny_Do_Pop",
           o_Zajetosc_Nieb          := "Wozek_Nieb_Zajetosc");
NETWORK
TITLE = Zezwolenie do poprzedniej
//Przypisanie bitow wyjsciowych
      A     "Wozek_zasprzeglony";
      JCN   kon;
//******************Zasprzeglenie KB1 *********************************
      A     "Zasprzeglenie_KB1";
      JCN   ekb1;
//***Zabierz do nastepnej
      A     "Wozek_Zabierz_Do_Nast";
      CLR;
//***Zezwolenie do poprzedniej
      A     "Wozek_Zez_Do_Pop";
      =     "DB_CONECTOR_KB1".Shuttle.Zez_Do_Pop;
//*** Paleta dostarczona do poprzedniej
      A     "Wozek_Paleta_Dost_Do_Pop";
      =     "DB_CONECTOR_KB1".Shuttle.Paleta_Dost_do_Pop;
//***Zezwolenie reczny do nastepniej
      A     "Wozek_Zez_Reczny_Do_Nast";
      CLR;
//***Zezwolenie reczny do przedniej
      A     "Wozek_Zez_Reczny_Do_Pop";
      =     "DB_CONECTOR_KB1".Shuttle.Zez_Reczny_do_Pop;
//***Skok na koniec
      JU    et_1;
ekb1: NOP   0;
//******************Zasprzeglenie KB2 *********************************
      A     "Zasprzeglenie_KB2";
      JCN   ekb2;
//***Zabierz do nastepnej
      A     "Wozek_Zabierz_Do_Nast";
      CLR;
//***Zezwolenie do poprzedniej
      A     "Wozek_Zez_Do_Pop";
      =     "DB_CONECTOR_KB2".Shuttle.Zez_Do_Pop;
//*** Paleta dostarczona do poprzedniej
      A     "Wozek_Paleta_Dost_Do_Pop";
      =     "DB_CONECTOR_KB2".Shuttle.Paleta_Dost_do_Pop;
//***Zezwolenie reczny do nastepniej
      A     "Wozek_Zez_Reczny_Do_Nast";
      CLR;
//***Zezwolenie reczny do przedniej
      A     "Wozek_Zez_Reczny_Do_Pop";
      =     "DB_CONECTOR_KB2".Shuttle.Zez_Reczny_do_Pop;
//***Skok na koniec
      JU    et_1;
ekb2: NOP   0;
//******************Zasprzeglenie pobierania I1 *********************************
      A     "Zasprzeglenie_Pob_I1";
      JCN   epob;
//***Zabierz do nastepnej
      A     "Wozek_Zabierz_Do_Nast";
      CLR;
//***Zezwolenie do poprzedniej
      A     "Wozek_Zez_Do_Pop";
      =     "DB_CONNECTOR_BUFF".Banda_I1_Shuttle.Zez_Do_Pop;
//*** Paleta dostarczona do poprzedniej
      A     "Wozek_Paleta_Dost_Do_Pop";
      =     "DB_CONNECTOR_BUFF".Banda_I1_Shuttle.Paleta_Dost_do_Pop;
//***Zezwolenie reczny do nastepniej
      A     "Wozek_Zez_Reczny_Do_Nast";
      CLR;
//***Zezwolenie reczny do przedniej
      A     "Wozek_Zez_Reczny_Do_Pop";
      =     "DB_CONNECTOR_BUFF".Banda_I1_Shuttle.Zez_Reczny_do_Pop;
//***Skok na koniec
      JU    et_1;
epob: NOP   0;
//******************Zasprzeglenie gender *********************************
      A     "Zasprzeglenie_Gender";
      JCN   egen;
//***Zabierz do nastepnej
      A     "Wozek_Zabierz_Do_Nast";
      =     "COM_GENDER".OUT.Wozek_Zab_do_Nast;
//***Zezwolenie do poprzedniej
      A     "Wozek_Zez_Do_Pop";
      CLR;
//*** Paleta dostarczona do poprzedniej
      A     "Wozek_Paleta_Dost_Do_Pop";
      CLR;
//***Zezwolenie reczny do nastepniej
      A     "Wozek_Zez_Reczny_Do_Nast";
      =     "COM_GENDER".OUT.Wozek_Zez_R_do_Nast;
//***Zezwolenie reczny do przedniej
      A     "Wozek_Zez_Reczny_Do_Pop";
      CLR;
//***Skok na koniec
      JU    et_1;
egen: NOP   0;
//******************Zasprzeglenie odbierania *********************************
      A     "Zasprzeglenie_Odbieranie";
      JCN   eodb;
//***Zabierz do nastepnej
      A     "Wozek_Zabierz_Do_Nast";
      =     "DB_CONNECTOR_BUFF".Banda_O1_Shuttle.Zabierz_do_Nast;
//***Zezwolenie do poprzedniej
      A     "Wozek_Zez_Do_Pop";
      CLR;
//*** Paleta dostarczona do poprzedniej
      A     "Wozek_Paleta_Dost_Do_Pop";
      CLR;
//***Zezwolenie reczny do nastepniej
      A     "Wozek_Zez_Reczny_Do_Nast";
      =     "DB_CONNECTOR_BUFF".Banda_O1_Shuttle.Zez_Reczny_do_Nast;
//***Zezwolenie reczny do przedniej
      A     "Wozek_Zez_Reczny_Do_Pop";
      CLR;
//***Skok na koniec
      JU    et_1;
eodb: NOP   0;
//******************Zasprzeglenie pobierania I2 *********************************
      A     "Zasprzeglenie_Pob_I2";
      JCN   e_I2;
//***Zabierz do nastepnej
      A     "Wozek_Zabierz_Do_Nast";
      CLR;
//***Zezwolenie do poprzedniej
      A     "Wozek_Zez_Do_Pop";
      =     "DB_CONNECTOR_BUFF".Banda_I2_Shuttle.Zez_Do_Pop;
//*** Paleta dostarczona do poprzedniej
      A     "Wozek_Paleta_Dost_Do_Pop";
      =     "DB_CONNECTOR_BUFF".Banda_I2_Shuttle.Paleta_Dost_do_Pop;
//***Zezwolenie reczny do nastepniej
      A     "Wozek_Zez_Reczny_Do_Nast";
      =     "DB_CONNECTOR_BUFF".Banda_I2_Shuttle.Zez_Reczny_do_Nast;
//***Zezwolenie reczny do przedniej
      A     "Wozek_Zez_Reczny_Do_Pop";
      =     "DB_CONNECTOR_BUFF".Banda_I2_Shuttle.Zez_Reczny_do_Pop;
//***Skok na koniec
      JU    et_1;
e_I2: NOP   0;
//******************Zasprzeglenie pobierania I3 *********************************
      A     "Zasprzeglenie_Pob_I3";
      JCN   e_I3;
//***Zabierz do nastepnej
      A     "Wozek_Zabierz_Do_Nast";
      CLR;
//***Zezwolenie do poprzedniej
      A     "Wozek_Zez_Do_Pop";
      =     "DB_CONNECTOR_BUFF".Banda_I3_Shuttle.Zez_Do_Pop;
//*** Paleta dostarczona do poprzedniej
      A     "Wozek_Paleta_Dost_Do_Pop";
      =     "DB_CONNECTOR_BUFF".Banda_I3_Shuttle.Paleta_Dost_do_Pop;
//***Zezwolenie reczny do nastepniej
      A     "Wozek_Zez_Reczny_Do_Nast";
      =     "DB_CONNECTOR_BUFF".Banda_I3_Shuttle.Zez_Reczny_do_Nast;
//***Zezwolenie reczny do przedniej
      A     "Wozek_Zez_Reczny_Do_Pop";
      =     "DB_CONNECTOR_BUFF".Banda_I3_Shuttle.Zez_Reczny_do_Pop;
//***Skok na koniec
      JU    et_1;
e_I3: NOP   0;
kon:  NOP   0;
//******************Wozek rozprzeglony *********************************
      SET;
      R     "DB_CONECTOR_KB1".Shuttle.Zez_Do_Pop;
      R     "DB_CONECTOR_KB1".Shuttle.Paleta_Dost_do_Pop;
      R     "DB_CONECTOR_KB1".Shuttle.Zez_Reczny_do_Pop;
      R     "DB_CONECTOR_KB2".Shuttle.Zez_Do_Pop;
      R     "DB_CONECTOR_KB2".Shuttle.Paleta_Dost_do_Pop;
      R     "DB_CONECTOR_KB2".Shuttle.Zez_Reczny_do_Pop;
      R     "DB_CONNECTOR_BUFF".Banda_I1_Shuttle.Zez_Do_Pop;
      R     "DB_CONNECTOR_BUFF".Banda_I1_Shuttle.Zez_Reczny_do_Pop;
      R     "DB_CONNECTOR_BUFF".Banda_I1_Shuttle.Paleta_Dost_do_Pop;
      R     "DB_CONNECTOR_BUFF".Banda_O1_Shuttle.Zabierz_do_Nast;
      R     "DB_CONNECTOR_BUFF".Banda_O1_Shuttle.Zez_Reczny_do_Nast;
      R     "COM_GENDER".OUT.Wozek_Zab_do_Nast;
      R     "COM_GENDER".OUT.Wozek_Zez_R_do_Nast;
      R     "DB_CONNECTOR_BUFF".Banda_I2_Shuttle.Zez_Do_Pop;
      R     "DB_CONNECTOR_BUFF".Banda_I2_Shuttle.Zez_Reczny_do_Pop;
      R     "DB_CONNECTOR_BUFF".Banda_I2_Shuttle.Paleta_Dost_do_Pop;
      R     "DB_CONNECTOR_BUFF".Banda_I3_Shuttle.Zez_Do_Pop;
      R     "DB_CONNECTOR_BUFF".Banda_I3_Shuttle.Zez_Reczny_do_Pop;
      R     "DB_CONNECTOR_BUFF".Banda_I3_Shuttle.Paleta_Dost_do_Pop;
//-Reset bitoow wychodzacych
      R     "Wozek_Zabierz_Do_Nast";
      R     "Wozek_Zez_Do_Pop";
      R     "Wozek_Paleta_Dost_Do_Pop";
      R     "Wozek_Zez_Reczny_Do_Nast";
      R     "Wozek_Zez_Reczny_Do_Pop";
      R     "Wozek_Nieb_Zajetosc";
//gender
//kb1
et_1: NOP   0;
END_FUNCTION_BLOCK

FUNCTION_BLOCK "Stanowisko_KB1"	// FB 3
//wyglad lini
//
//
//||||   ||     ||||   ||||
//|Z||  |O||    |W |   |S |
//||||   ||     ||||   ||||
//      
//      ||||
//      |B||
//      ||||
//
//Gdzie:
//-W-Winda
//-S-Shuttle
//-Z-ZPA(Segbert)
//-O-Obrotnica
//-B-Banda Backup
//
//
//Wersja 1.1
//-Dodanie mo¿liwosci poboru palety z Bandy backup (pisanie w trakcie)
//
//
//
AUTHOR : Kng
NAME : KB1
VERSION : 0.1
VAR
  KB1_Wylot_2 : FB 33;
  KB1_Obrotnica : FB 35;
  KB1_Uzbrajanie : FB 10;
  KB1_Winda : FB 37;
END_VAR
BEGIN
NETWORK
TITLE =
//Ten Network celowo jest wolny
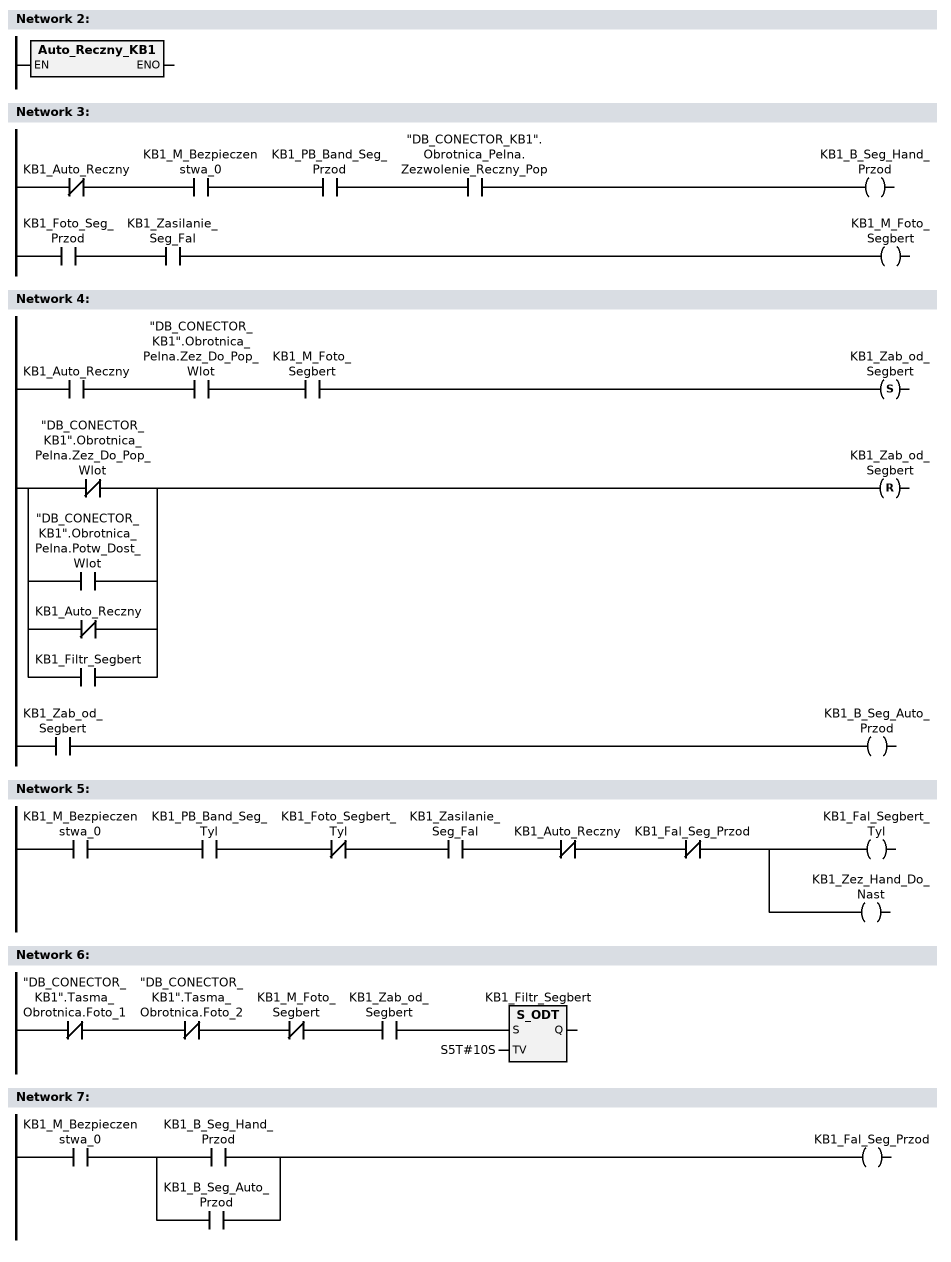
NETWORK
TITLE =
      CALL  "Auto_Reczny_KB1";
      NOP   0;
NETWORK
TITLE =
//Bity do Terminala
//
//Terminal_Palet                                   Szafa_Transport
//
//
//<-----------------------------------------------KB2_Fal_Seg_Przod (Q25.0)
//<-----------------------------------------------
//<-----------------------------------------------
//
//----------------------------------------------->KB2_Foto_Seg_Przod (I26.0)
//----------------------------------------------->
//----------------------------------------------->
//----------------------------------------------->
      AN    "KB1_Auto_Reczny";
      A     "KB1_M_Bezpieczenstwa_0";
      A     "KB1_PB_Band_Seg_Przod";
      A     "DB_CONECTOR_KB1".Obrotnica_Pelna.Zezwolenie_Reczny_Pop;
      =     "KB1_B_Seg_Hand_Przod";
//Wyjazd palety w automacie
      A     "KB1_Foto_Seg_Przod";
      A     "KB1_Zasilanie_Seg_Fal";
      =     "KB1_M_Foto_Segbert";
NETWORK
TITLE =
      A     "KB1_Auto_Reczny";
      A     "DB_CONECTOR_KB1".Obrotnica_Pelna.Zez_Do_Pop_Wlot;
      A     "KB1_M_Foto_Segbert";
      S     "KB1_Zab_od_Segbert";
      A(;
      ON    "DB_CONECTOR_KB1".Obrotnica_Pelna.Zez_Do_Pop_Wlot;
      O     "DB_CONECTOR_KB1".Obrotnica_Pelna.Potw_Dost_Wlot;
      ON    "KB1_Auto_Reczny";
      O     "KB1_Filtr_Segbert";
      );
      R     "KB1_Zab_od_Segbert";
      A     "KB1_Zab_od_Segbert";
      =     "KB1_B_Seg_Auto_Przod";
NETWORK
TITLE =
//Segbert_Warunkowy tyl
      A     "KB1_M_Bezpieczenstwa_0";
      A     "KB1_PB_Band_Seg_Tyl";
      AN    "KB1_Foto_Segbert_Tyl";
      A     "KB1_Zasilanie_Seg_Fal";
      AN    "KB1_Auto_Reczny";
      AN    "KB1_Fal_Seg_Przod";
      =     "KB1_Fal_Segbert_Tyl";
      =     "KB1_Zez_Hand_Do_Nast";
NETWORK
TITLE =
      AN    "DB_CONECTOR_KB1".Tasma_Obrotnica.Foto_1;
      AN    "DB_CONECTOR_KB1".Tasma_Obrotnica.Foto_2;
      AN    "KB1_M_Foto_Segbert";
      A     "KB1_Zab_od_Segbert";
      L     S5T#10S;
      SD    "KB1_Filtr_Segbert";
      NOP   0;
      NOP   0;
      NOP   0;
      NOP   0;
NETWORK
TITLE =
//Jazda bandy Segbert do przodu
      A     "KB1_M_Bezpieczenstwa_0";
      A(;
      O     "KB1_B_Seg_Hand_Przod";
      O     "KB1_B_Seg_Auto_Przod";
      );
      =     "KB1_Fal_Seg_Przod";
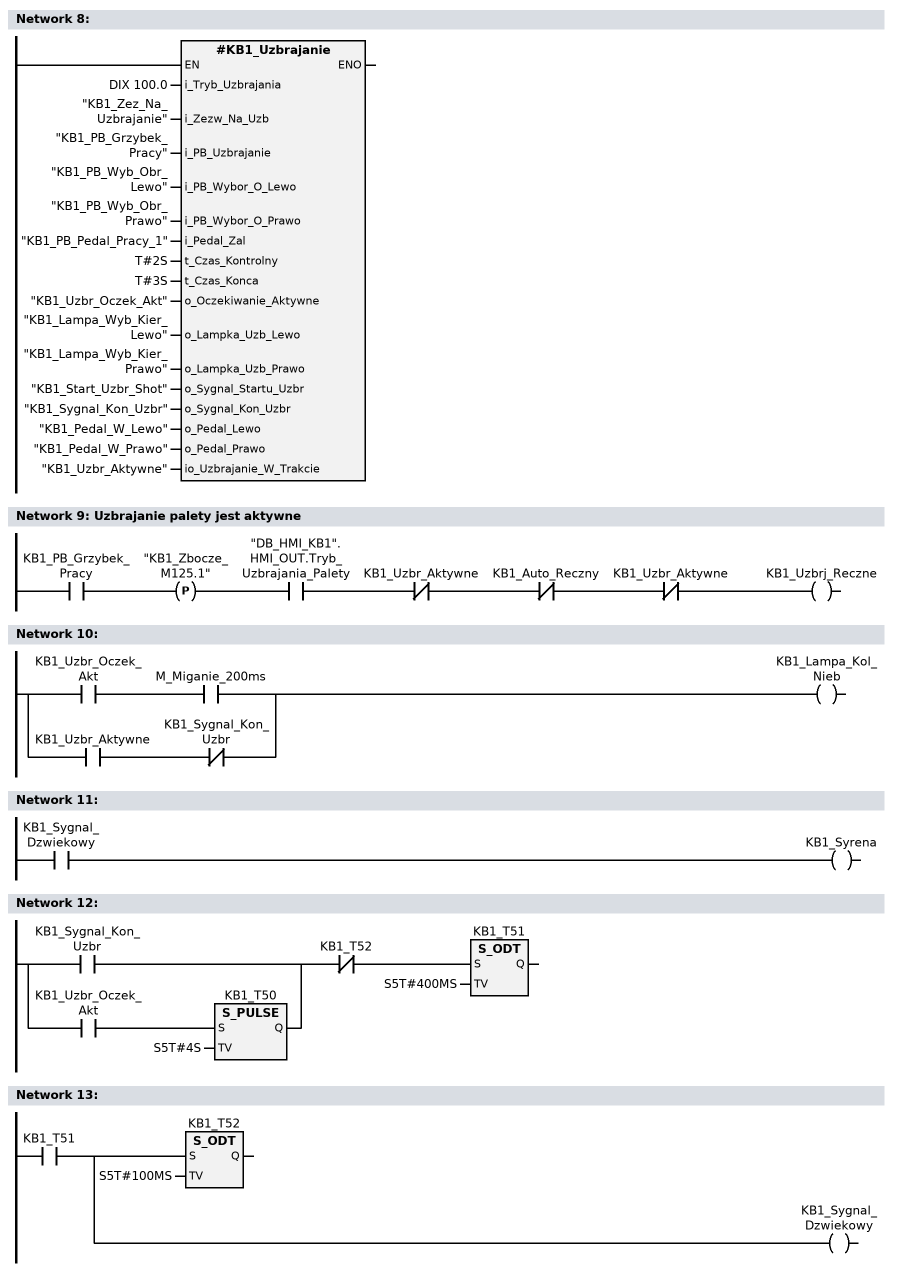
NETWORK
TITLE =
//Funkcja Uzbrajania
      CALL  #KB1_Uzbrajanie (
           i_Tryb_Uzbrajania        := DIX 100.0,
           i_Zezw_Na_Uzb            := "KB1_Zez_Na_Uzbrajanie",
           i_PB_Uzbrajanie          := "KB1_PB_Grzybek_Pracy",
           i_PB_Wybor_O_Lewo        := "KB1_PB_Wyb_Obr_Lewo",
           i_PB_Wybor_O_Prawo       := "KB1_PB_Wyb_Obr_Prawo",
           i_Pedal_Zal              := "KB1_PB_Pedal_Pracy_1",
           t_Czas_Kontrolny         := T#2S,
           t_Czas_Konca             := T#3S,
           o_Oczekiwanie_Aktywne    := "KB1_Uzbr_Oczek_Akt",
           o_Lampka_Uzb_Lewo        := "KB1_Lampa_Wyb_Kier_Lewo",
           o_Lampka_Uzb_Prawo       := "KB1_Lampa_Wyb_Kier_Prawo",
           o_Sygnal_Startu_Uzbr     := "KB1_Start_Uzbr_Shot",
           o_Sygnal_Kon_Uzbr        := "KB1_Sygnal_Kon_Uzbr",
           o_Pedal_Lewo             := "KB1_Pedal_W_Lewo",
           o_Pedal_Prawo            := "KB1_Pedal_W_Prawo",
           io_Uzbrajanie_W_Trakcie  := "KB1_Uzbr_Aktywne");
NETWORK
TITLE = Uzbrajanie palety jest aktywne
//Uzbrajanie reczne 
      A     "KB1_PB_Grzybek_Pracy";
      FP    "KB1_Zbocze_M125.1";
      A     "DB_HMI_KB1".HMI_OUT.Tryb_Uzbrajania_Palety;
      AN    "KB1_Uzbr_Aktywne";
      AN    "KB1_Auto_Reczny";
      AN    "KB1_Uzbr_Aktywne";
      =     "KB1_Uzbrj_Reczne";
NETWORK
TITLE =
//Lampka uzbrajania
//
      A     "KB1_Uzbr_Oczek_Akt";
      A     "M_Miganie_200ms";
      O;
      A     "KB1_Uzbr_Aktywne";
      AN    "KB1_Sygnal_Kon_Uzbr";
      =     "KB1_Lampa_Kol_Nieb";
NETWORK
TITLE =
//Sygnal dzwiekowy uzbrajania
//
      A     "KB1_Sygnal_Dzwiekowy";
      =     "KB1_Syrena";
NETWORK
TITLE =
//Tworzenie dzwieku
      A(;
      O     "KB1_Sygnal_Kon_Uzbr";
      O(;
      A     "KB1_Uzbr_Oczek_Akt";
      L     S5T#4S;
      SP    "KB1_T50";
      NOP   0;
      NOP   0;
      NOP   0;
      A     "KB1_T50";
      );
      );
      AN    "KB1_T52";
      L     S5T#400MS;
      SD    "KB1_T51";
      NOP   0;
      NOP   0;
      NOP   0;
      NOP   0;
NETWORK
TITLE =
      A     "KB1_T51";
      =     L 0.0;
      A     L 0.0;
      L     S5T#100MS;
      SD    "KB1_T52";
      NOP   0;
      NOP   0;
      NOP   0;
      NOP   0;
      A     L 0.0;
      BLD   102;
      =     "KB1_Sygnal_Dzwiekowy";
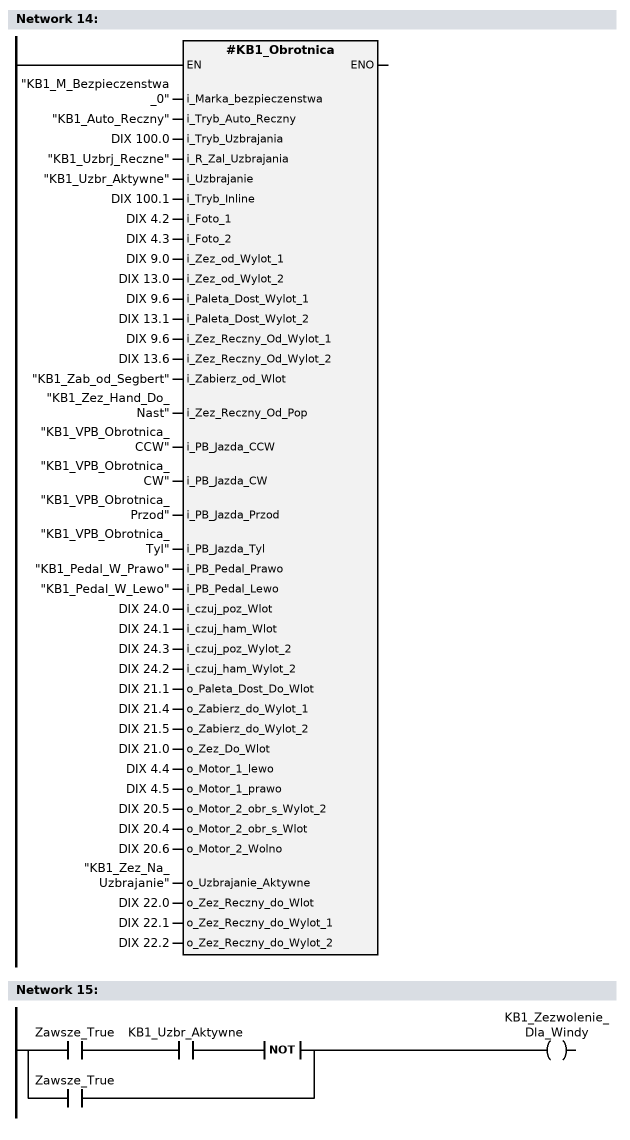
NETWORK
TITLE =
//Obrotnica z funkcja uzbrajania
      CALL  #KB1_Obrotnica (
           i_Marka_bezpieczenstwa   := "KB1_M_Bezpieczenstwa_0",
           i_Tryb_Auto_Reczny       := "KB1_Auto_Reczny",
           i_Tryb_Uzbrajania        := DIX 100.0,
           i_R_Zal_Uzbrajania       := "KB1_Uzbrj_Reczne",
           i_Uzbrajanie             := "KB1_Uzbr_Aktywne",
           i_Tryb_Inline            := DIX 100.1,
           i_Foto_1                 := DIX 4.2,
           i_Foto_2                 := DIX 4.3,
           i_Zez_od_Wylot_1         := DIX 9.0,
           i_Zez_od_Wylot_2         := DIX 13.0,
           i_Paleta_Dost_Wylot_1    := DIX 9.6,
           i_Paleta_Dost_Wylot_2    := DIX 13.1,
           i_Zez_Reczny_Od_Wylot_1  := DIX 9.6,
           i_Zez_Reczny_Od_Wylot_2  := DIX 13.6,
           i_Zabierz_od_Wlot        := "KB1_Zab_od_Segbert",
           i_Zez_Reczny_Od_Pop      := "KB1_Zez_Hand_Do_Nast",
           i_PB_Jazda_CCW           := "KB1_VPB_Obrotnica_CCW",
           i_PB_Jazda_CW            := "KB1_VPB_Obrotnica_CW",
           i_PB_Jazda_Przod         := "KB1_VPB_Obrotnica_Przod",
           i_PB_Jazda_Tyl           := "KB1_VPB_Obrotnica_Tyl",
           i_PB_Pedal_Prawo         := "KB1_Pedal_W_Prawo",
           i_PB_Pedal_Lewo          := "KB1_Pedal_W_Lewo",
           i_czuj_poz_Wlot          := DIX 24.0,
           i_czuj_ham_Wlot          := DIX 24.1,
           i_czuj_poz_Wylot_2       := DIX 24.3,
           i_czuj_ham_Wylot_2       := DIX 24.2,
           o_Paleta_Dost_Do_Wlot    := DIX 21.1,
           o_Zabierz_do_Wylot_1     := DIX 21.4,
           o_Zabierz_do_Wylot_2     := DIX 21.5,
           o_Zez_Do_Wlot            := DIX 21.0,
           o_Motor_1_lewo           := DIX 4.4,
           o_Motor_1_prawo          := DIX 4.5,
           o_Motor_2_obr_s_Wylot_2  := DIX 20.5,
           o_Motor_2_obr_s_Wlot     := DIX 20.4,
           o_Motor_2_Wolno          := DIX 20.6,
           o_Uzbrajanie_Aktywne     := "KB1_Zez_Na_Uzbrajanie",
           o_Zez_Reczny_do_Wlot     := DIX 22.0,
           o_Zez_Reczny_do_Wylot_1  := DIX 22.1,
           o_Zez_Reczny_do_Wylot_2  := DIX 22.2);
NETWORK
TITLE =
      A     "Zawsze_True";
      A     "KB1_Uzbr_Aktywne";
      NOT;
      O     "Zawsze_True";
      =     "KB1_Zezwolenie_Dla_Windy";
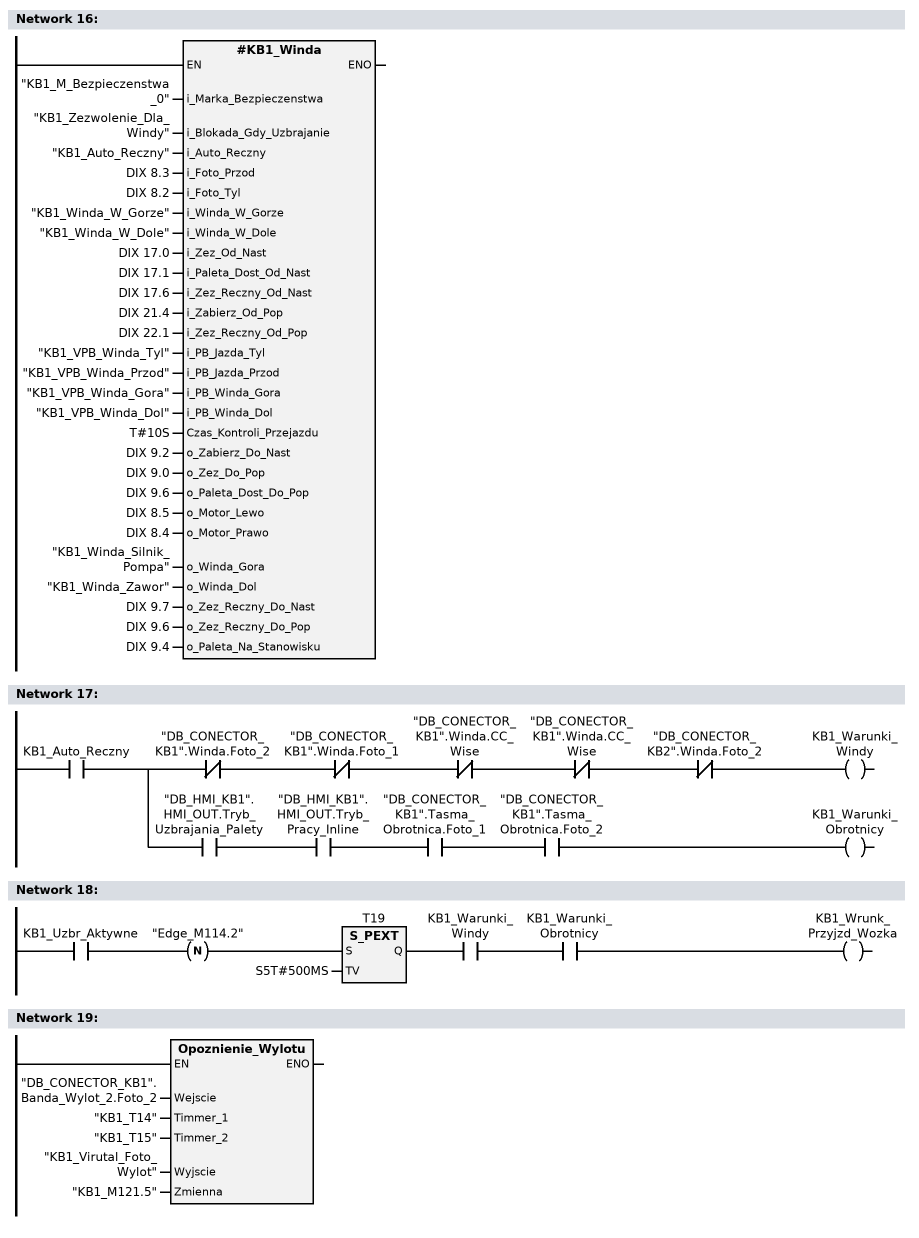
NETWORK
TITLE =
//Winda
      CALL  #KB1_Winda (
           i_Marka_Bezpieczenstwa   := "KB1_M_Bezpieczenstwa_0",
           i_Blokada_Gdy_Uzbrajanie := "KB1_Zezwolenie_Dla_Windy",
           i_Auto_Reczny            := "KB1_Auto_Reczny",
           i_Foto_Przod             := DIX 8.3,
           i_Foto_Tyl               := DIX 8.2,
           i_Winda_W_Gorze          := "KB1_Winda_W_Gorze",
           i_Winda_W_Dole           := "KB1_Winda_W_Dole",
           i_Zez_Od_Nast            := DIX 17.0,
           i_Paleta_Dost_Od_Nast    := DIX 17.1,
           i_Zez_Reczny_Od_Nast     := DIX 17.6,
           i_Zabierz_Od_Pop         := DIX 21.4,
           i_Zez_Reczny_Od_Pop      := DIX 22.1,
           i_PB_Jazda_Tyl           := "KB1_VPB_Winda_Tyl",
           i_PB_Jazda_Przod         := "KB1_VPB_Winda_Przod",
           i_PB_Winda_Gora          := "KB1_VPB_Winda_Gora",
           i_PB_Winda_Dol           := "KB1_VPB_Winda_Dol",
           Czas_Kontroli_Przejazdu  := T#10S,
           o_Zabierz_Do_Nast        := DIX 9.2,
           o_Zez_Do_Pop             := DIX 9.0,
           o_Paleta_Dost_Do_Pop     := DIX 9.6,
           o_Motor_Lewo             := DIX 8.5,
           o_Motor_Prawo            := DIX 8.4,
           o_Winda_Gora             := "KB1_Winda_Silnik_Pompa",
           o_Winda_Dol              := "KB1_Winda_Zawor",
           o_Zez_Reczny_Do_Nast     := DIX 9.7,
           o_Zez_Reczny_Do_Pop      := DIX 9.6,
           o_Paleta_Na_Stanowisku   := DIX 9.4);
NETWORK
TITLE =
//Warunkowa jazda wozka gdy konczone jest owijanie
//Warunki windy.
      A     "KB1_Auto_Reczny";
      =     L 0.0;
      A     L 0.0;
      AN    "DB_CONECTOR_KB1".Winda.Foto_2;
      AN    "DB_CONECTOR_KB1".Winda.Foto_1;
      AN    "DB_CONECTOR_KB1".Winda.CC_Wise;
      AN    "DB_CONECTOR_KB1".Winda.CC_Wise;
      AN    "DB_CONECTOR_KB2".Winda.Foto_2;
      =     "KB1_Warunki_Windy";
      A     L 0.0;
      A     "DB_HMI_KB1".HMI_OUT.Tryb_Uzbrajania_Palety;
      A     "DB_HMI_KB1".HMI_OUT.Tryb_Pracy_Inline;
      A     "DB_CONECTOR_KB1".Tasma_Obrotnica.Foto_1;
      A     "DB_CONECTOR_KB1".Tasma_Obrotnica.Foto_2;
      =     "KB1_Warunki_Obrotnicy";
NETWORK
TITLE =
//Warunki obrotnicy
      A(;
      A     "KB1_Uzbr_Aktywne";
      FN    "Edge_M114.2";
      L     S5T#500MS;
      SE    "T19";
      NOP   0;
      NOP   0;
      NOP   0;
      A     "T19";
      );
      A     "KB1_Warunki_Windy";
      A     "KB1_Warunki_Obrotnicy";
      =     "KB1_Wrunk_Przyjzd_Wozka";
NETWORK
TITLE =
//Opoznienie wylotu
      CALL  "Opoznienie_Wylotu" (
           Wejscie                  := "DB_CONECTOR_KB1".Banda_Wylot_2.Foto_2,
           Timmer_1                 := "KB1_T14",
           Timmer_2                 := "KB1_T15",
           Wyjscie                  := "KB1_Virutal_Foto_Wylot",
           Zmienna                  := "KB1_M121.5");
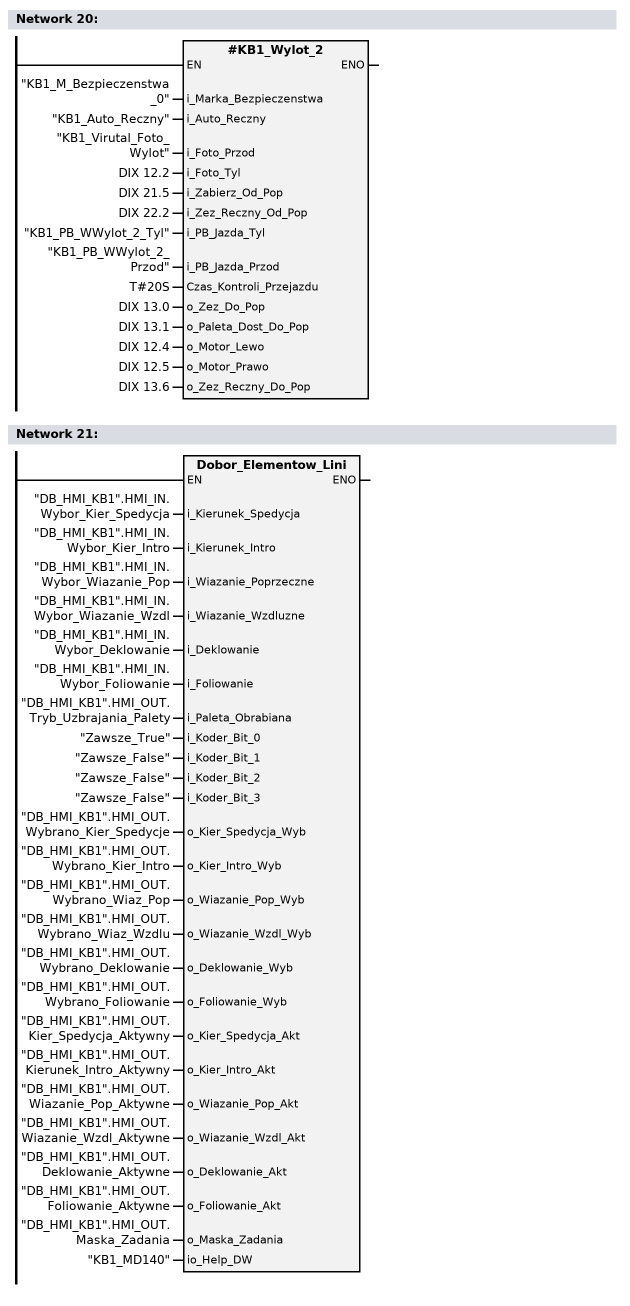
NETWORK
TITLE =
//Banda Wylot 2
      CALL  #KB1_Wylot_2 (
           i_Marka_Bezpieczenstwa   := "KB1_M_Bezpieczenstwa_0",
           i_Auto_Reczny            := "KB1_Auto_Reczny",
           i_Foto_Przod             := "KB1_Virutal_Foto_Wylot",
           i_Foto_Tyl               := DIX 12.2,
           i_Zabierz_Od_Pop         := DIX 21.5,
           i_Zez_Reczny_Od_Pop      := DIX 22.2,
           i_PB_Jazda_Tyl           := "KB1_PB_WWylot_2_Tyl",
           i_PB_Jazda_Przod         := "KB1_PB_WWylot_2_Przod",
           Czas_Kontroli_Przejazdu  := T#20S,
           o_Zez_Do_Pop             := DIX 13.0,
           o_Paleta_Dost_Do_Pop     := DIX 13.1,
           o_Motor_Lewo             := DIX 12.4,
           o_Motor_Prawo            := DIX 12.5,
           o_Zez_Reczny_Do_Pop      := DIX 13.6);
NETWORK
TITLE =
//fc400. Kod kolbus 2 to 2 .
      CALL  "Dobor_Elementow_Lini" (
           i_Kierunek_Spedycja      := "DB_HMI_KB1".HMI_IN.Wybor_Kier_Spedycja,
           i_Kierunek_Intro         := "DB_HMI_KB1".HMI_IN.Wybor_Kier_Intro,
           i_Wiazanie_Poprzeczne    := "DB_HMI_KB1".HMI_IN.Wybor_Wiazanie_Pop,
           i_Wiazanie_Wzdluzne      := "DB_HMI_KB1".HMI_IN.Wybor_Wiazanie_Wzdl,
           i_Deklowanie             := "DB_HMI_KB1".HMI_IN.Wybor_Deklowanie,
           i_Foliowanie             := "DB_HMI_KB1".HMI_IN.Wybor_Foliowanie,
           i_Paleta_Obrabiana       := "DB_HMI_KB1".HMI_OUT.Tryb_Uzbrajania_Palety,
           i_Koder_Bit_0            := "Zawsze_True",
           i_Koder_Bit_1            := "Zawsze_False",
           i_Koder_Bit_2            := "Zawsze_False",
           i_Koder_Bit_3            := "Zawsze_False",
           o_Kier_Spedycja_Wyb      := "DB_HMI_KB1".HMI_OUT.Wybrano_Kier_Spedycje,
           o_Kier_Intro_Wyb         := "DB_HMI_KB1".HMI_OUT.Wybrano_Kier_Intro,
           o_Wiazanie_Pop_Wyb       := "DB_HMI_KB1".HMI_OUT.Wybrano_Wiaz_Pop,
           o_Wiazanie_Wzdl_Wyb      := "DB_HMI_KB1".HMI_OUT.Wybrano_Wiaz_Wzdlu,
           o_Deklowanie_Wyb         := "DB_HMI_KB1".HMI_OUT.Wybrano_Deklowanie,
           o_Foliowanie_Wyb         := "DB_HMI_KB1".HMI_OUT.Wybrano_Foliowanie,
           o_Kier_Spedycja_Akt      := "DB_HMI_KB1".HMI_OUT.Kier_Spedycja_Aktywny,
           o_Kier_Intro_Akt         := "DB_HMI_KB1".HMI_OUT.Kierunek_Intro_Aktywny,
           o_Wiazanie_Pop_Akt       := "DB_HMI_KB1".HMI_OUT.Wiazanie_Pop_Aktywne,
           o_Wiazanie_Wzdl_Akt      := "DB_HMI_KB1".HMI_OUT.Wiazanie_Wzdl_Aktywne,
           o_Deklowanie_Akt         := "DB_HMI_KB1".HMI_OUT.Deklowanie_Aktywne,
           o_Foliowanie_Akt         := "DB_HMI_KB1".HMI_OUT.Foliowanie_Aktywne,
           o_Maska_Zadania          := "DB_HMI_KB1".HMI_OUT.Maska_Zadania,
           io_Help_DW               := "KB1_MD140");
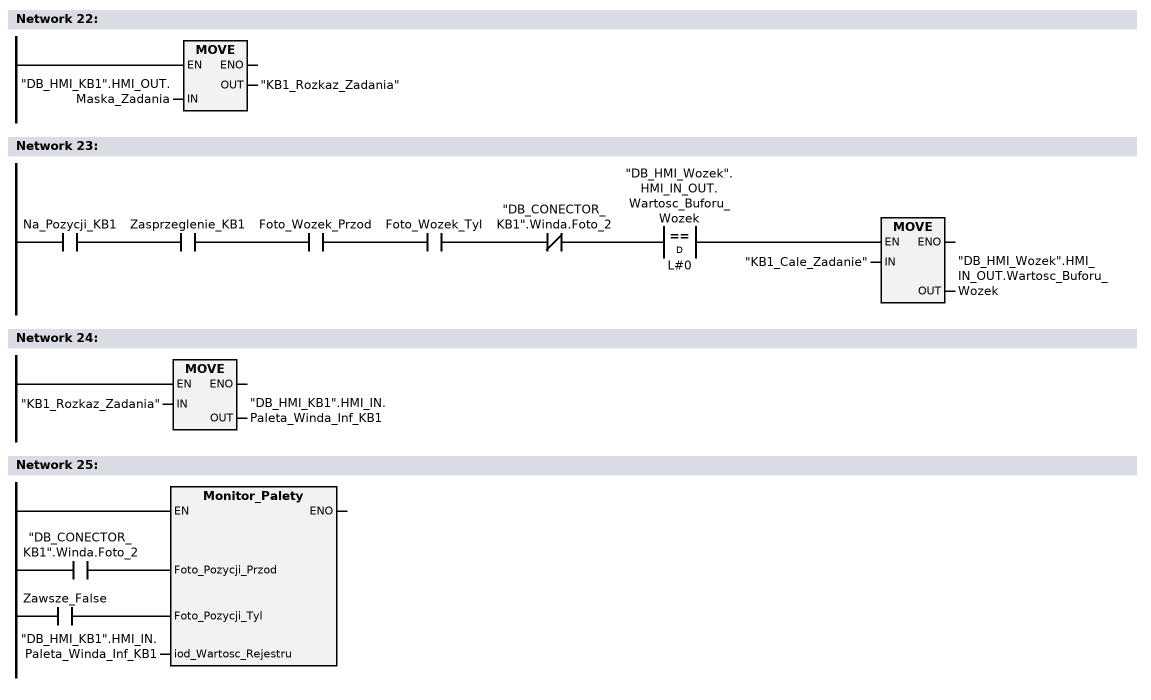
NETWORK
TITLE =
//Przeslanie maski do starszego slowa
      L     "DB_HMI_KB1".HMI_OUT.Maska_Zadania;
      T     "KB1_Rozkaz_Zadania";
      NOP   0;
NETWORK
TITLE =
//To jest wozek
//
      A     "Na_Pozycji_KB1";
      A     "Zasprzeglenie_KB1";
      A     "Foto_Wozek_Przod";
      A     "Foto_Wozek_Tyl";
      AN    "DB_CONECTOR_KB1".Winda.Foto_2;
      A(;
      L     "DB_HMI_Wozek".HMI_IN_OUT.Wartosc_Buforu_Wozek;
      L     L#0;
      ==D;
      );
      JNB   _001;
      L     "KB1_Cale_Zadanie";
      T     "DB_HMI_Wozek".HMI_IN_OUT.Wartosc_Buforu_Wozek;
_001: NOP   0;
NETWORK
TITLE =
      L     "KB1_Rozkaz_Zadania";
      T     "DB_HMI_KB1".HMI_IN.Paleta_Winda_Inf_KB1;
      NOP   0;
NETWORK
TITLE =
      A     "DB_CONECTOR_KB1".Winda.Foto_2;
      =     L 0.0;
      BLD   103;
      A     "Zawsze_False";
      =     L 0.1;
      BLD   103;
      CALL  "Monitor_Palety" (
           Foto_Pozycji_Przod       := L 0.0,
           Foto_Pozycji_Tyl         := L 0.1,
           iod_Wartosc_Rejestru     := "DB_HMI_KB1".HMI_IN.Paleta_Winda_Inf_KB1);
      NOP   0;
END_FUNCTION_BLOCK

